(***************************判断纠偏从轴1是否超限********************************)	
AxisRecDevPos_H:=arrAxisPar[SlaveNo1].arrTargetPoint[0]-AxisPos_H;//轴纠偏上限
AxisRecDevPos_L:=arrAxisPar[SlaveNo1].arrTargetPoint[0]-AxisPos_L;//轴纠偏下限
AxisRecDevActPos1:=REAL_TO_LREAL(arrAxisCtrl[SlaveNo1].Status.fActPos);
IF AxisRecDevActPos1 > AxisRecDevPos_H OR AxisRecDevActPos1 < AxisRecDevPos_L THEN
	PosOverLimit1:=TRUE;//纠偏超限
ELSE
	PosOverLimit1:=FALSE;
END_IF
(***************************判断纠偏从轴2是否超限********************************)	
AxisRecDevPos_H:=arrAxisPar[SlaveNo2].arrTargetPoint[0]-AxisPos_H;//轴纠偏上限
AxisRecDevPos_L:=arrAxisPar[SlaveNo2].arrTargetPoint[0]-AxisPos_L;//轴纠偏下限
AxisRecDevActPos2:=REAL_TO_LREAL(arrAxisCtrl[SlaveNo2].Status.fActPos);
IF AxisRecDevActPos2 > AxisRecDevPos_H OR AxisRecDevActPos2 < AxisRecDevPos_L THEN
	PosOverLimit1:=TRUE;//纠偏超限
ELSE
	PosOverLimit1:=FALSE;
END_IF

IF Enable THEN
	CASE Step0 OF
		0://判断凸轮是否耦合
			IF NOT TON2.Q THEN
				TON2.IN:=TRUE;
				IF arrAxisCtrl[SlaveNo1].Status.Coupled AND arrAxisCtrl[SlaveNo2].Status.Coupled  THEN
					TON2.IN:=FALSE;
					Step0:=10;					
				END_IF
			ELSE
					TON2.IN:=FALSE;
					Error[0]:=TRUE;//纠偏凸轮耦合失败
					Step0:=9999;	//报警	
			END_IF
		10://判断主轴是是否启动，没启动则启动主轴
				IF arrAxisCtrl[MasterNo].Status.fActVelo>0 THEN
					Step0:=20;
				ELSE
					arrAxisCtrl[MasterNo].Cmd.bEnable:=TRUE;
					IF arrAxisCtrl[MasterNo].Status.Enabled THEN
						arrAxisPar[MasterNo].fVelocity_of_Velo:=MasterValue;//主轴速度
						arrAxisCtrl[MasterNo].Cmd.bMoveVelo:=TRUE;//主轴匀速启动							
					END_IF
				END_IF
		20://从轴纠偏速度计算
				TON1.IN:=TRUE;		
				IF RecDevPV > RecDevSensors_H AND TON1.Q THEN //纠偏传感器的当前值 大于 纠偏上限 
					IF NOT PosOverLimit1 AND NOT  PosOverLimit2 AND  arrAxisCtrl[SlaveNo1].Io.biNegLimit  AND  arrAxisCtrl[SlaveNo2].Io.biNegLimit  THEN//判断纠偏是否超限
						MC_RecDevvelocity_M:=(RecDevPV-RecDevSensors_H)*RecDevSpeedCoe;
						IF NOT CWW THEN
							MC_RecDevvelocity:=ScaleTrans(EN:=TRUE , Scalln:=MC_RecDevvelocity_M , X0:=0 , Y0:=0 , X1:=400 , Y1:=10 , Sclofs:=0 );//ScaleTrans的作用是将X0至X1范围之间的输入值，转换为Y0至Y1范围之间的输出值
						ELSE
							MC_RecDevvelocity:=-ScaleTrans(EN:=TRUE , Scalln:=MC_RecDevvelocity_M , X0:=0 , Y0:=0 , X1:=400 , Y1:=10 , Sclofs:=0 );
						END_IF
					ELSE
						Error[1]:=TRUE;//纠偏负限位报警
						MC_RecDevvelocity:=0;
					END_IF
				ELSIF RecDevPV < RecDevSensors_L AND TON1.Q  THEN//纠偏传感器的当前值 小于 纠偏下限
					IF NOT PosOverLimit1 AND NOT PosOverLimit2 AND  arrAxisCtrl[SlaveNo1].Io.biPosLimit AND  arrAxisCtrl[SlaveNo2].Io.biPosLimit  THEN
						MC_RecDevvelocity_M:=(RecDevSensors_L-RecDevPV)*RecDevSpeedCoe;//判断纠偏是否超限
						IF NOT CWW THEN
							MC_RecDevvelocity:=-ScaleTrans(EN:=TRUE , Scalln:=MC_RecDevvelocity_M , X0:=0 , Y0:=0 , X1:=400 , Y1:=10 , Sclofs:=0 );
						ELSE
							MC_RecDevvelocity:=ScaleTrans(EN:=TRUE , Scalln:=MC_RecDevvelocity_M , X0:=0 , Y0:=0 , X1:=400 , Y1:=10 , Sclofs:=0 );
						END_IF	
					ELSE
						Error[2]:=TRUE;//纠偏正限位报警
						MC_RecDevvelocity:=0;
					END_IF	
				ELSE
					MC_RecDevvelocity:=0;		
				END_IF					
	END_CASE
ELSE
		MC_RecDevvelocity:=0;//从轴的纠偏速度
		Step0:=0;
		TON1.IN:=FALSE;
		TON2.IN:=FALSE;
		IF RestHMI THEN
			Error[0]:=FALSE;//纠偏凸轮耦合失败
			Error[1]:=FALSE;//纠偏负限位报警
			Error[2]:=FALSE;//纠偏正限位报警
		END_IF
END_IF	
//纠偏齿轮耦合
IF MasterValue<>0 THEN
	GearInMultiMaster.GearRatio1:=MC_RecDevvelocity/MasterValue;
ELSE
	GearInMultiMaster.GearRatio1:=0;
END_IF
//多主轴耦合，不管主轴的停止还是运行中，都可以耦合从轴
GearInMultiMaster(
	Master1:=arrAxis[MasterNo] , 
	Master2:=arrAxis[SlaveNo1] , 
	Master3:=arrAxis[SlaveNo1] , 
	Master4:=arrAxis[SlaveNo1] , 
	Slave:=arrAxis[SlaveNo1]  , 
	Enable:=Enable , 
	GearRatio1:= , 
	GearRatio2:=0 , 
	GearRatio3:=0 , 
	GearRatio4:=0 , 
	Acceleration:= , 
	Deceleration:= , 
	Jerk:= , 
	BufferMode:= , 
	Options:= , 
	InGear=> , 
	Busy=> , 
	Active=> , 
	CommandAborted=> , 
	Error=> , 
	ErrorID=> );
//多主轴耦合，不管主轴的停止还是运行中，都可以耦合从轴
GearInMultiMaster1(
	Master1:=arrAxis[SlaveNo1] , 
	Master2:=arrAxis[SlaveNo2] , 
	Master3:=arrAxis[SlaveNo2] , 
	Master4:=arrAxis[SlaveNo2] , 
	Slave:=arrAxis[SlaveNo2]  , 
	Enable:=Enable , 
	GearRatio1:=1 , 
	GearRatio2:=0 , 
	GearRatio3:=0 , 
	GearRatio4:=0 , 
	Acceleration:= , 
	Deceleration:= , 
	Jerk:= , 
	BufferMode:= , 
	Options:= , 
	InGear=> , 
	Busy=> , 
	Active=> , 
	CommandAborted=> , 
	Error=> , 
	ErrorID=> );	
//纠偏从轴1解耦
SlaveCamOut(
	Slave:=arrAxis[SlaveNo1] , 
	Execute:=sF_TRIG.Q OR sR_TRIG.Q , 
	Options:= , 
	Done=> , 
	Busy=> , 
	Error=> , 
	ErrorID=> );
	//纠偏从轴2解耦
SlaveCamOut2(
	Slave:=arrAxis[SlaveNo2] , 
	Execute:=sF_TRIG.Q OR sR_TRIG.Q , 
	Options:= , 
	Done=> , 
	Busy=> , 
	Error=> , 
	ErrorID=> );
//从轴1停止
Slave_Stop(
	Axis:=arrAxis[SlaveNo1] , 
	Execute:=sF_TRIG.Q   , 
	Deceleration:= , 
	Jerk:= , 
	Options:= , 
	Done=> , 
	Busy=> , 
	Active=> , 
	CommandAborted=> , 
	Error=> , 
	ErrorID=> );
//从轴2停止
Slave_Stop2(
	Axis:=arrAxis[SlaveNo2] , 
	Execute:=sF_TRIG.Q   , 
	Deceleration:= , 
	Jerk:= , 
	Options:= , 
	Done=> , 
	Busy=> , 
	Active=> , 
	CommandAborted=> , 
	Error=> , 
	ErrorID=> );

END_FUNCTION_BLOCK

// ---- P2POUs/BasicFunction/01_IO/ScaleTrans.TcPOU
FUNCTION ScaleTrans : REAL
VAR_INPUT
	EN:BOOL;//启动条件
	Scalln:REAL;//输入值
	X0:REAL;//输入范围下限值
	Y0:REAL;//输出范围下限值
	X1:REAL;//输入范围上限值
	Y1:REAL;//输出范围上限值
	Sclofs:REAL;//偏置值
END_VAR
VAR
END_VAR

IF EN THEN
	IF (X1-X0)<> 0 THEN
		ScaleTrans:=(Y1-Y0)/(X1-X0)*(Scalln-X0)+Y0+Sclofs;
	END_IF
END_IF

END_FUNCTION

// ---- P2POUs/BasicFunction/12_User2/FB_BlueGlue.TcPOU
FUNCTION_BLOCK FB_BlueGlue//蓝胶检测自动
VAR_INPUT
	Enable:BOOL;//启动条件
	BlueSenser:BOOL;//蓝胶检测信号
	An_Quantited:UINT;//正极已叠片极片数
	An_QuantitSet:UINT;//正极设定叠片片
	Ca_Quantited:UINT;//负极已叠片极片数
	Ca_QuantitSet:UINT;//负极设定叠片片
	Distance:REAL;//蓝胶检测Semer到压刀的距离
	BluWidth:REAL;//蓝胶宽度
	Width:REAL;//压刀外边距宽度	 
END_VAR
VAR_OUTPUT
END_VAR
VAR_IN_OUT
		BluGlueNG:ARRAY[0..1] OF BOOL;
END_VAR
VAR
	// 正、负极已叠极片总数
	Quantited: UINT;
	// 正、负极设定极片总数
	QuantitSet: UINT;
	// 正、负极未叠片数
	Quantit: UINT;
	// 未叠极片所需隔膜长度
	Distance_DT: REAL;
	// 蓝胶到压刀距离上限
	Distance_H: REAL;
	// 蓝胶到压针距离下限
	Distance_L: REAL;
	Step0: INT;

	blue_R_TRIG: R_TRIG;
	blue_F_TRIG: F_TRIG;
END_VAR

//计算已叠极片总数
Quantited:=An_Quantited+Ca_Quantited;
//计算正、负极片设定总数
QuantitSet:=An_QuantitSet+Ca_QuantitSet;
//计算未叠片数
Quantit:=QuantitSet-Quantited;
//未叠正、负极片所需隔膜总长度
Distance_DT:=Width*Quantit;
//蓝胶到压针距离上限
Distance_H:=Distance+BluWidth+10;
//蓝胶到压针距离下降
Distance_L:=Distance+BluWidth-10;
//蓝胶检测信号上升沿
blue_R_TRIG(CLK:=BlueSenser, Q=> );
//蓝胶要信号下降沿
blue_F_TRIG(CLK:=BlueSenser , Q=> );
IF Enable THEN
	CASE Step0 OF
			0://判断是否检测到蓝胶信号
				IF blue_R_TRIG.Q THEN
					Step0:=10;
				END_IF
			10://根据未叠片隔膜长度与蓝胶到压刀的距离判断是当前电芯NG、下一个电芯NG、当前以及下一个电芯都NG
				IF  Distance_DT<Distance_L THEN //未叠片隔膜长度小于蓝胶所需隔膜长度下限，下一个电芯NG
					BluGlueNG[1]:=TRUE;
					Step0:=20;
				ELSIF Distance_DT>Distance_L AND Distance_DT< Distance_H  THEN//未叠片隔膜长度在蓝胶上、下限之间，则当前电芯、下个电芯都NG
					BluGlueNG[0]:=TRUE;
					BluGlueNG[1]:=TRUE;
					Step0:=20;
				ELSIF Distance_DT> Distance_H THEN//未叠片隔膜长度大于蓝胶所需隔膜长度上限，当前电芯NG
					BluGlueNG[0]:=TRUE;
					Step0:=20;
				END_IF
			20://判断检测是否结束
				IF blue_F_TRIG.Q THEN
					Step0:=0;
				END_IF
	END_CASE
END_IF

END_FUNCTION_BLOCK

// ---- P2POUs/BasicFunction/12_User2/FB_Demarcate.TcPOU
FUNCTION_BLOCK FB_Demarcate//CCD标定自动程序
VAR_INPUT
	AxisX1_NO : INT; //X1轴号
	AxisX2_NO : INT;//X2轴号
	AxisY_NO  : INT;//Y轴号	
END_VAR
VAR_OUTPUT
	
END_VAR
VAR
	
	i: INT;
	// 拍照延时复位
	TON1: TON;
	TON2: TON;
	// CCD标定上升沿
	rCCD_Demarcate: R_TRIG;
	singeMode: BOOL;
	singeStep0: BOOL;
	fCCD_Demarcate: F_TRIG;
	bTest1: BOOL;
	iTest: INT;
END_VAR

VAR_IN_OUT
	Step0: INT;//程序步
	DemarcateStart:BOOL;//CCD标定启动	
	CCDStart: BOOL;// CCD拍照启动
	CCDNo:INT;//ccd拍照次数记数
	DemarcateResult:INT;//标定结果
	DemarcateDone: BOOL;	// CCD标定完成
	Demarcateing: BOOL;	// CCD标定中
	// CCD标定NG报警
	Error: BOOL;
END_VAR

TON1(IN:= , PT:=T#2S , Q=> , ET=> );//拍照延时复位
TON2(IN:= , PT:=T#0.2S , Q=> , ET=> );//拍照延时
rCCD_Demarcate(CLK:=DemarcateStart , Q=> );//CCD标定启动上升沿
fCCD_Demarcate(CLK:=DemarcateStart , Q=> );//CCD标定启动上升沿
IF rCCD_Demarcate.Q THEN
	Error:=FALSE;//CCD标定NG报警
	TON1.IN:=FALSE;
	Step0:=0;
END_IF



CASE Step0 OF
		0://等待CCD标定启动信号
			IF fCCD_Demarcate.Q THEN
						i:=0;//标定点位记数
						TON1.IN:=FALSE;
						DemarcateStart:=FALSE;//复位标定启动
						DemarcateDone:=FALSE;//CCD标定完成
						Demarcateing:=TRUE;//CCD标定中
						IF singeMode THEN
							singeStep0:=TRUE;
						ELSE
							singeStep0:=FALSE;
						END_IF
						Step0:=10;
			END_IF
	10://X1、X2先回初始位
				IF  NOT singeStep0 THEN
							TON1.IN:=FALSE;
							IF arrAxisCtrl[AxisX1_NO].Status.Homed AND arrAxisCtrl[AxisX1_NO].Status.NoMoving THEN
										IF arrAxisCtrl[AxisX1_NO].Cmd.arrbRealPoint[1] THEN
											arrAxisCtrl[AxisX1_NO].Cmd.iGoSetPos:=0;
										ELSE
											arrAxisCtrl[AxisX1_NO].Cmd.iGoSetPos:=1;
										END_IF
							END_IF
							IF arrAxisCtrl[AxisX2_NO].Status.Homed AND arrAxisCtrl[AxisX2_NO].Status.NoMoving  THEN
										IF arrAxisCtrl[AxisX2_NO].Cmd.arrbRealPoint[1] THEN
											arrAxisCtrl[AxisX2_NO].Cmd.iGoSetPos:=0;
										ELSE
											arrAxisCtrl[AxisX2_NO].Cmd.iGoSetPos:=1;
										END_IF
							END_IF	
							IF  arrAxisCtrl[AxisX1_NO].Cmd.arrbRealPoint[1]  AND 	arrAxisCtrl[AxisX2_NO].Cmd.arrbRealPoint[1]THEN
								IF singeMode THEN
									singeStep0:=TRUE;
								ELSE
									singeStep0:=FALSE;
								END_IF
								Step0:=11;
							END_IF	
				END_IF		
	11://Y回初始位
				IF NOT singeStep0 THEN
									IF arrAxisCtrl[AxisY_NO].Status.Homed AND arrAxisCtrl[AxisY_NO].Status.NoMoving  THEN
											IF arrAxisCtrl[AxisY_NO].Cmd.arrbRealPoint[1] THEN
												arrAxisCtrl[AxisY_NO].Cmd.iGoSetPos:=0;
													IF singeMode THEN
														singeStep0:=TRUE;
													ELSE
														singeStep0:=FALSE;
													END_IF
													Step0:=12;									
											ELSE
												arrAxisCtrl[AxisY_NO].Cmd.iGoSetPos:=1;
											END_IF
								END_IF
				END_IF			
		12://判断CCD标定走到第几个点位
						IF NOT  singeStep0 THEN
											DemarcateResult:=0;
											IF  i=0    THEN//(-4,-4)
															arrAxisPar[AxisX1_NO].arrTargetPoint[3]:=arrAxisPar[AxisX1_NO].arrTargetPoint[1]-4;//+(103.94*COS(DEG_TO_RAD(CCD_W+225))-103.94*COS(DEG_TO_RAD(225))); 
															arrAxisPar[AxisX2_NO].arrTargetPoint[3]:=arrAxisPar[AxisX2_NO].arrTargetPoint[1]-4;//+(103.94*SIN(DEG_TO_RAD(CCD_W+315))-103.94*COS(DEG_TO_RAD(315)));
															arrAxisPar[AxisY_NO].arrTargetPoint[3]:=arrAxisPar[AxisY_NO].arrTargetPoint[1]-4;//+(103.94*COS(DEG_TO_RAD(CCD_W+135))-103.94*COS(DEG_TO_RAD(135)));	
															i:=i+1;
															IF singeMode THEN
																singeStep0:=TRUE;
															ELSE
																singeStep0:=FALSE;
															END_IF
															Step0:=20;
											ELSIF i=1 THEN//(0,-4)
															arrAxisPar[AxisX1_NO].arrTargetPoint[3]:=arrAxisPar[AxisX1_NO].arrTargetPoint[1];//+(103.94*COS(DEG_TO_RAD(CCD_W+225))-103.94*COS(DEG_TO_RAD(225))); 
															arrAxisPar[AxisX2_NO].arrTargetPoint[3]:=arrAxisPar[AxisX2_NO].arrTargetPoint[1];//+(103.94*SIN(DEG_TO_RAD(CCD_W+315))-103.94*COS(DEG_TO_RAD(315)));
															arrAxisPar[AxisY_NO].arrTargetPoint[3]:=arrAxisPar[AxisY_NO].arrTargetPoint[1]-4;//+(103.94*COS(DEG_TO_RAD(CCD_W+135))-103.94*COS(DEG_TO_RAD(135)));
															i:=i+1;
															IF singeMode THEN
																singeStep0:=TRUE;
															ELSE
																singeStep0:=FALSE;
															END_IF
															Step0:=20;
											ELSIF i=2 THEN//(4,-4)
															arrAxisPar[AxisX1_NO].arrTargetPoint[3]:=arrAxisPar[AxisX1_NO].arrTargetPoint[1]+4;//+(103.94*COS(DEG_TO_RAD(CCD_W+225))-103.94*COS(DEG_TO_RAD(225))); 
															arrAxisPar[AxisX2_NO].arrTargetPoint[3]:=arrAxisPar[AxisX2_NO].arrTargetPoint[1]+4;//+(103.94*SIN(DEG_TO_RAD(CCD_W+315))-103.94*COS(DEG_TO_RAD(315)));
															arrAxisPar[AxisY_NO].arrTargetPoint[3]:=arrAxisPar[AxisY_NO].arrTargetPoint[1]-4;//+(103.94*COS(DEG_TO_RAD(CCD_W+135))-103.94*COS(DEG_TO_RAD(135)));	
															i:=i+1;
															IF singeMode THEN
																singeStep0:=TRUE;
															ELSE
																singeStep0:=FALSE;
															END_IF
															Step0:=20;									
											ELSIF i=3 THEN//(4,0)
														arrAxisPar[AxisX1_NO].arrTargetPoint[3]:=arrAxisPar[AxisX1_NO].arrTargetPoint[1]+4;//+(103.94*COS(DEG_TO_RAD(CCD_W+225))-103.94*COS(DEG_TO_RAD(225))); 
														arrAxisPar[AxisX2_NO].arrTargetPoint[3]:=arrAxisPar[AxisX2_NO].arrTargetPoint[1]+4;//+(103.94*SIN(DEG_TO_RAD(CCD_W+315))-103.94*COS(DEG_TO_RAD(315)));
														arrAxisPar[AxisY_NO].arrTargetPoint[3]:=arrAxisPar[AxisY_NO].arrTargetPoint[1];//+(103.94*COS(DEG_TO_RAD(CCD_W+135))-103.94*COS(DEG_TO_RAD(135)));	
														i:=i+1;
														IF singeMode THEN
																singeStep0:=TRUE;
															ELSE
																singeStep0:=FALSE;
															END_IF
														Step0:=20;		
											ELSIF i=4 THEN//(0,0)
														arrAxisPar[AxisX1_NO].arrTargetPoint[3]:=arrAxisPar[AxisX1_NO].arrTargetPoint[1];//+(103.94*COS(DEG_TO_RAD(CCD_W+225))-103.94*COS(DEG_TO_RAD(225))); 
														arrAxisPar[AxisX2_NO].arrTargetPoint[3]:=arrAxisPar[AxisX2_NO].arrTargetPoint[1];//+(103.94*SIN(DEG_TO_RAD(CCD_W+315))-103.94*COS(DEG_TO_RAD(315)));
														arrAxisPar[AxisY_NO].arrTargetPoint[3]:=arrAxisPar[AxisY_NO].arrTargetPoint[1];//+(103.94*COS(DEG_TO_RAD(CCD_W+135))-103.94*COS(DEG_TO_RAD(135)));	
														i:=i+1;
														Step0:=20;		
											ELSIF i=5 THEN//(-4,0)
														arrAxisPar[AxisX1_NO].arrTargetPoint[3]:=arrAxisPar[AxisX1_NO].arrTargetPoint[1]-4;//+(103.94*COS(DEG_TO_RAD(CCD_W+225))-103.94*COS(DEG_TO_RAD(225))); 
														arrAxisPar[AxisX2_NO].arrTargetPoint[3]:=arrAxisPar[AxisX2_NO].arrTargetPoint[1]-4;//+(103.94*SIN(DEG_TO_RAD(CCD_W+315))-103.94*COS(DEG_TO_RAD(315)));
														arrAxisPar[AxisY_NO].arrTargetPoint[3]:=arrAxisPar[AxisY_NO].arrTargetPoint[1];//+(103.94*COS(DEG_TO_RAD(CCD_W+135))-103.94*COS(DEG_TO_RAD(135)));	
														i:=i+1;
														IF singeMode THEN
																singeStep0:=TRUE;
															ELSE
																singeStep0:=FALSE;
															END_IF
														Step0:=20;		
											ELSIF i=6 THEN//(-4,4)
															arrAxisPar[AxisX1_NO].arrTargetPoint[3]:=arrAxisPar[AxisX1_NO].arrTargetPoint[1]-4;//+(103.94*COS(DEG_TO_RAD(CCD_W+225))-103.94*COS(DEG_TO_RAD(225))); 
															arrAxisPar[AxisX2_NO].arrTargetPoint[3]:=arrAxisPar[AxisX2_NO].arrTargetPoint[1]-4;//+(103.94*SIN(DEG_TO_RAD(CCD_W+315))-103.94*COS(DEG_TO_RAD(315)));
															arrAxisPar[AxisY_NO].arrTargetPoint[3]:=arrAxisPar[AxisY_NO].arrTargetPoint[1]+4;//+(103.94*COS(DEG_TO_RAD(CCD_W+135))-103.94*COS(DEG_TO_RAD(135)));
															i:=i+1;
															IF singeMode THEN
																singeStep0:=TRUE;
															ELSE
																singeStep0:=FALSE;
															END_IF
															Step0:=20;		
											ELSIF i=7 THEN//(0,4)
															arrAxisPar[AxisX1_NO].arrTargetPoint[3]:=arrAxisPar[AxisX1_NO].arrTargetPoint[1];//+(103.94*COS(DEG_TO_RAD(CCD_W+225))-103.94*COS(DEG_TO_RAD(225))); 
															arrAxisPar[AxisX2_NO].arrTargetPoint[3]:=arrAxisPar[AxisX2_NO].arrTargetPoint[1];//+(103.94*SIN(DEG_TO_RAD(CCD_W+315))-103.94*COS(DEG_TO_RAD(315)));
															arrAxisPar[AxisY_NO].arrTargetPoint[3]:=arrAxisPar[AxisY_NO].arrTargetPoint[1]+4;//+(103.94*COS(DEG_TO_RAD(CCD_W+135))-103.94*COS(DEG_TO_RAD(135)));	
															i:=i+1;
															IF singeMode THEN
																singeStep0:=TRUE;
															ELSE
																singeStep0:=FALSE;
															END_IF
															Step0:=20;		
											ELSIF i=8 THEN//(4,4)
														arrAxisPar[AxisX1_NO].arrTargetPoint[3]:=arrAxisPar[AxisX1_NO].arrTargetPoint[1]+4;//+(103.94*COS(DEG_TO_RAD(CCD_W+225))-103.94*COS(DEG_TO_RAD(225))); 
														arrAxisPar[AxisX2_NO].arrTargetPoint[3]:=arrAxisPar[AxisX2_NO].arrTargetPoint[1]+4;//+(103.94*SIN(DEG_TO_RAD(CCD_W+315))-103.94*COS(DEG_TO_RAD(315)));
														arrAxisPar[AxisY_NO].arrTargetPoint[3]:=arrAxisPar[AxisY_NO].arrTargetPoint[1]+4;//+(103.94*COS(DEG_TO_RAD(CCD_W+135))-103.94*COS(DEG_TO_RAD(135)));	
														i:=i+1;
														IF singeMode THEN
																singeStep0:=TRUE;
															ELSE
																singeStep0:=FALSE;
															END_IF
														Step0:=20;		
											ELSIF i=9 THEN//(0,0,-2)
														arrAxisPar[AxisX1_NO].arrTargetPoint[3]:=arrAxisPar[AxisX1_NO].arrTargetPoint[1]+(103.94*COS(DEG_TO_RAD(-2+225))-103.94*COS(DEG_TO_RAD(225))); 
														arrAxisPar[AxisX2_NO].arrTargetPoint[3]:=arrAxisPar[AxisX2_NO].arrTargetPoint[1]+(103.94*COS(DEG_TO_RAD(-2+135))-103.94*COS(DEG_TO_RAD(135)));
														arrAxisPar[AxisY_NO].arrTargetPoint[3]:=arrAxisPar[AxisY_NO].arrTargetPoint[1]+(103.94*SIN(DEG_TO_RAD(-2+315))-103.94*SIN(DEG_TO_RAD(315)));	
														i:=i+1;
														IF singeMode THEN
																singeStep0:=TRUE;
															ELSE
																singeStep0:=FALSE;
															END_IF
														Step0:=20;		
											ELSIF i=10 THEN//(0,0)
														arrAxisPar[AxisX1_NO].arrTargetPoint[3]:=arrAxisPar[AxisX1_NO].arrTargetPoint[1];//+(103.94*COS(DEG_TO_RAD(2+225))-103.94*COS(DEG_TO_RAD(225))); 
														arrAxisPar[AxisX2_NO].arrTargetPoint[3]:=arrAxisPar[AxisX2_NO].arrTargetPoint[1];//+(103.94*SIN(DEG_TO_RAD(2+315))-103.94*COS(DEG_TO_RAD(315)));
														arrAxisPar[AxisY_NO].arrTargetPoint[3]:=arrAxisPar[AxisY_NO].arrTargetPoint[1];//+(103.94*COS(DEG_TO_RAD(2+135))-103.94*COS(DEG_TO_RAD(135)));	
														i:=i+1;
														IF singeMode THEN
																singeStep0:=TRUE;
															ELSE
																singeStep0:=FALSE;
															END_IF
														Step0:=20;		
											ELSIF i=11  THEN//(0,0,2)
															arrAxisPar[AxisX1_NO].arrTargetPoint[3]:=arrAxisPar[AxisX1_NO].arrTargetPoint[1]+(103.94*COS(DEG_TO_RAD(2+225))-103.94*COS(DEG_TO_RAD(225))); 
															arrAxisPar[AxisX2_NO].arrTargetPoint[3]:=arrAxisPar[AxisX2_NO].arrTargetPoint[1]+(103.94*COS(DEG_TO_RAD(2+135))-103.94*COS(DEG_TO_RAD(135)));
															arrAxisPar[AxisY_NO].arrTargetPoint[3]:=arrAxisPar[AxisY_NO].arrTargetPoint[1]+(103.94*SIN(DEG_TO_RAD(2+315))-103.94*SIN(DEG_TO_RAD(315)));
															i:=i+1;
															IF singeMode THEN
																singeStep0:=TRUE;
															ELSE
																singeStep0:=FALSE;
															END_IF
															Step0:=20;		
											ELSIF i=130 THEN
															arrAxisPar[AxisX1_NO].arrTargetPoint[3]:=arrAxisPar[AxisX1_NO].arrTargetPoint[1];//+(103.94*COS(DEG_TO_RAD(CCD_W+225))-103.94*COS(DEG_TO_RAD(225))); 
															arrAxisPar[AxisX2_NO].arrTargetPoint[3]:=arrAxisPar[AxisX2_NO].arrTargetPoint[1];//+(103.94*SIN(DEG_TO_RAD(CCD_W+315))-103.94*COS(DEG_TO_RAD(315)));
															arrAxisPar[AxisY_NO].arrTargetPoint[3]:=arrAxisPar[AxisY_NO].arrTargetPoint[1];//+(103.94*COS(DEG_TO_RAD(CCD_W+135))-103.94*COS(DEG_TO_RAD(135)));	
															i:=i+1;
															IF singeMode THEN
																singeStep0:=TRUE;
															ELSE
																singeStep0:=FALSE;
															END_IF
															Step0:=20;		
											ELSIF i=140 THEN
														arrAxisPar[AxisX1_NO].arrTargetPoint[3]:=arrAxisPar[AxisX1_NO].arrTargetPoint[1]+(103.94*COS(DEG_TO_RAD(-1+225))-103.94*COS(DEG_TO_RAD(225))); 
														arrAxisPar[AxisX2_NO].arrTargetPoint[3]:=arrAxisPar[AxisX2_NO].arrTargetPoint[1]+(103.94*SIN(DEG_TO_RAD(-1+315))-103.94*COS(DEG_TO_RAD(315)));
														arrAxisPar[AxisY_NO].arrTargetPoint[3]:=arrAxisPar[AxisY_NO].arrTargetPoint[1]+(103.94*COS(DEG_TO_RAD(-1+135))-103.94*COS(DEG_TO_RAD(135)));	
														i:=i+1;
														IF singeMode THEN
																singeStep0:=TRUE;
															ELSE
																singeStep0:=FALSE;
															END_IF
														Step0:=20;		
											ELSIF i=150 THEN
														arrAxisPar[AxisX1_NO].arrTargetPoint[3]:=arrAxisPar[AxisX1_NO].arrTargetPoint[1]+(103.94*COS(DEG_TO_RAD(-2+225))-103.94*COS(DEG_TO_RAD(225))); 
														arrAxisPar[AxisX2_NO].arrTargetPoint[3]:=arrAxisPar[AxisX2_NO].arrTargetPoint[1]+(103.94*SIN(DEG_TO_RAD(-2+315))-103.94*COS(DEG_TO_RAD(315)));
														arrAxisPar[AxisY_NO].arrTargetPoint[3]:=arrAxisPar[AxisY_NO].arrTargetPoint[1]+(103.94*COS(DEG_TO_RAD(-2+135))-103.94*COS(DEG_TO_RAD(135)));	
														i:=i+1;
														IF singeMode THEN
																singeStep0:=TRUE;
															ELSE
																singeStep0:=FALSE;
															END_IF
														Step0:=20;		
											ELSIF i=160 THEN
														arrAxisPar[AxisX1_NO].arrTargetPoint[3]:=arrAxisPar[AxisX1_NO].arrTargetPoint[1];//+(103.94*COS(DEG_TO_RAD(CCD_W+225))-103.94*COS(DEG_TO_RAD(225))); 
														arrAxisPar[AxisX2_NO].arrTargetPoint[3]:=arrAxisPar[AxisX2_NO].arrTargetPoint[1];//+(103.94*SIN(DEG_TO_RAD(CCD_W+315))-103.94*COS(DEG_TO_RAD(315)));
														arrAxisPar[AxisY_NO].arrTargetPoint[3]:=arrAxisPar[AxisY_NO].arrTargetPoint[1];//+(103.94*COS(DEG_TO_RAD(CCD_W+135))-103.94*COS(DEG_TO_RAD(135)));		
														i:=i+1;
														Step0:=20;													
											END_IF
						END_IF	
	20://先移动X1,X2
				IF  NOT singeStep0 THEN
					IF NOT TON1.Q THEN
										TON1.IN:=TRUE;
					ELSE
										IF arrAxisCtrl[AxisX1_NO].Status.Homed AND arrAxisCtrl[AxisX1_NO].Status.NoMoving THEN
													IF arrAxisCtrl[AxisX1_NO].Cmd.arrbRealPoint[3] THEN
														arrAxisCtrl[AxisX1_NO].Cmd.iGoSetPos:=0;
													ELSE
														arrAxisCtrl[AxisX1_NO].Cmd.iGoSetPos:=3;
													END_IF
										END_IF
										IF arrAxisCtrl[AxisX2_NO].Status.Homed AND arrAxisCtrl[AxisX2_NO].Status.NoMoving  THEN
													IF arrAxisCtrl[AxisX2_NO].Cmd.arrbRealPoint[3] THEN
														arrAxisCtrl[AxisX2_NO].Cmd.iGoSetPos:=0;
													ELSE
														arrAxisCtrl[AxisX2_NO].Cmd.iGoSetPos:=3;
													END_IF
										END_IF	
										IF  arrAxisCtrl[AxisX1_NO].Cmd.arrbRealPoint[3]  AND arrAxisCtrl[AxisX1_NO].Status.NoMoving AND 
							 				arrAxisCtrl[AxisX2_NO].Cmd.arrbRealPoint[3] AND arrAxisCtrl[AxisX2_NO].Status.NoMoving THEN
													IF singeMode THEN
														singeStep0:=TRUE;
													ELSE
														singeStep0:=FALSE;
													END_IF
													TON1.IN:=FALSE;
													Step0:=30;
										ELSIF arrAxisCtrl[AxisX1_NO].Status.Error OR arrAxisCtrl[AxisX2_NO].Status.Error THEN
													TON1.IN:=FALSE;
													Step0:=0;											
										END_IF	
						END_IF
				END_IF	
	30://再移动Y
				IF NOT singeStep0 THEN
							IF NOT TON1.Q THEN
										TON1.IN:=TRUE;
							ELSE
									IF arrAxisCtrl[AxisY_NO].Status.Homed AND arrAxisCtrl[AxisY_NO].Status.NoMoving  THEN
												IF arrAxisCtrl[AxisY_NO].Cmd.arrbRealPoint[3] THEN
													arrAxisCtrl[AxisY_NO].Cmd.iGoSetPos:=0;
														IF singeMode THEN
															singeStep0:=TRUE;
														ELSE
															singeStep0:=FALSE;
														END_IF
														TON1.IN:=FALSE;
														 TON2.IN:=FALSE;
														Step0:=31;									
												ELSE
													arrAxisCtrl[AxisY_NO].Cmd.iGoSetPos:=3;
												END_IF
								ELSIF   arrAxisCtrl[AxisY_NO].Status.Error THEN
														TON1.IN:=FALSE;
														Step0:=0;										
								END_IF
							END_IF
				END_IF
				
	31:
	    TON2.IN:=TRUE;
		IF TON2.Q THEN
				CCDNo:=i;
				CCDStart:=TRUE;
				DemarcateResult:=0;	
				Step0:=40;	
				 TON2.IN:=FALSE;
		END_IF		 
	40://启动拍照
			IF NOT TON1.Q THEN
				TON1.IN:=TRUE;
			ELSE
				TON1.IN:=FALSE;	
				CCDStart:=FALSE;
				Step0:=50;
			END_IF
	50://等待标定结果
			IF DemarcateResult=1 THEN
				DemarcateResult:=0; 
				 Step0:=60;
			ELSE
				Error:=TRUE;//CCD标定NG报警
				Step0:=9999;
			END_IF
	60://判断标定次数
			IF i>=12 THEN
				Step0:=0;
				Demarcateing:=FALSE;
			ELSE
				Step0:=10;
			END_IF				
END_CASE







IF bTest1 THEN
	
   CASE iTest OF
	 0://(-4,-4)
				arrAxisPar[AxisX1_NO].arrTargetPoint[3]:=arrAxisPar[AxisX1_NO].arrTargetPoint[1]-4;//+(103.94*COS(DEG_TO_RAD(CCD_W+225))-103.94*COS(DEG_TO_RAD(225))); 
				arrAxisPar[AxisX2_NO].arrTargetPoint[3]:=arrAxisPar[AxisX2_NO].arrTargetPoint[1]-4;//+(103.94*SIN(DEG_TO_RAD(CCD_W+315))-103.94*COS(DEG_TO_RAD(315)));
				arrAxisPar[AxisY_NO].arrTargetPoint[3]:=arrAxisPar[AxisY_NO].arrTargetPoint[1]-4;//+(103.94*COS(DEG_TO_RAD(CCD_W+135))-103.94*COS(DEG_TO_RAD(135)));	
				iTest:=50;
											
	 1://(0,-4)
			arrAxisPar[AxisX1_NO].arrTargetPoint[3]:=arrAxisPar[AxisX1_NO].arrTargetPoint[1];//+(103.94*COS(DEG_TO_RAD(CCD_W+225))-103.94*COS(DEG_TO_RAD(225))); 
		    arrAxisPar[AxisX2_NO].arrTargetPoint[3]:=arrAxisPar[AxisX2_NO].arrTargetPoint[1];//+(103.94*SIN(DEG_TO_RAD(CCD_W+315))-103.94*COS(DEG_TO_RAD(315)));
			arrAxisPar[AxisY_NO].arrTargetPoint[3]:=arrAxisPar[AxisY_NO].arrTargetPoint[1]-4;//+(103.94*COS(DEG_TO_RAD(CCD_W+135))-103.94*COS(DEG_TO_RAD(135)));
				iTest:=50;											
	2://(4,-4)
			arrAxisPar[AxisX1_NO].arrTargetPoint[3]:=arrAxisPar[AxisX1_NO].arrTargetPoint[1]+4;//+(103.94*COS(DEG_TO_RAD(CCD_W+225))-103.94*COS(DEG_TO_RAD(225))); 
			arrAxisPar[AxisX2_NO].arrTargetPoint[3]:=arrAxisPar[AxisX2_NO].arrTargetPoint[1]+4;//+(103.94*SIN(DEG_TO_RAD(CCD_W+315))-103.94*COS(DEG_TO_RAD(315)));
			arrAxisPar[AxisY_NO].arrTargetPoint[3]:=arrAxisPar[AxisY_NO].arrTargetPoint[1]-4;//+(103.94*COS(DEG_TO_RAD(CCD_W+135))-103.94*COS(DEG_TO_RAD(135)));	
				iTest:=50;															
	3://(4,0)
			arrAxisPar[AxisX1_NO].arrTargetPoint[3]:=arrAxisPar[AxisX1_NO].arrTargetPoint[1]+4;//+(103.94*COS(DEG_TO_RAD(CCD_W+225))-103.94*COS(DEG_TO_RAD(225))); 
			arrAxisPar[AxisX2_NO].arrTargetPoint[3]:=arrAxisPar[AxisX2_NO].arrTargetPoint[1]+4;//+(103.94*SIN(DEG_TO_RAD(CCD_W+315))-103.94*COS(DEG_TO_RAD(315)));
			arrAxisPar[AxisY_NO].arrTargetPoint[3]:=arrAxisPar[AxisY_NO].arrTargetPoint[1];//+(103.94*COS(DEG_TO_RAD(CCD_W+135))-103.94*COS(DEG_TO_RAD(135)));	
			iTest:=50;								
  4://(0,0)
		arrAxisPar[AxisX1_NO].arrTargetPoint[3]:=arrAxisPar[AxisX1_NO].arrTargetPoint[1];//+(103.94*COS(DEG_TO_RAD(CCD_W+225))-103.94*COS(DEG_TO_RAD(225))); 
		arrAxisPar[AxisX2_NO].arrTargetPoint[3]:=arrAxisPar[AxisX2_NO].arrTargetPoint[1];//+(103.94*SIN(DEG_TO_RAD(CCD_W+315))-103.94*COS(DEG_TO_RAD(315)));
			arrAxisPar[AxisY_NO].arrTargetPoint[3]:=arrAxisPar[AxisY_NO].arrTargetPoint[1];//+(103.94*COS(DEG_TO_RAD(CCD_W+135))-103.94*COS(DEG_TO_RAD(135)));	
			iTest:=50;
5://(-4,0)
			arrAxisPar[AxisX1_NO].arrTargetPoint[3]:=arrAxisPar[AxisX1_NO].arrTargetPoint[1]-4;//+(103.94*COS(DEG_TO_RAD(CCD_W+225))-103.94*COS(DEG_TO_RAD(225))); 
			arrAxisPar[AxisX2_NO].arrTargetPoint[3]:=arrAxisPar[AxisX2_NO].arrTargetPoint[1]-4;//+(103.94*SIN(DEG_TO_RAD(CCD_W+315))-103.94*COS(DEG_TO_RAD(315)));
		arrAxisPar[AxisY_NO].arrTargetPoint[3]:=arrAxisPar[AxisY_NO].arrTargetPoint[1];//+(103.94*COS(DEG_TO_RAD(CCD_W+135))-103.94*COS(DEG_TO_RAD(135)));	
		iTest:=50;
6://(-4,4)
			arrAxisPar[AxisX1_NO].arrTargetPoint[3]:=arrAxisPar[AxisX1_NO].arrTargetPoint[1]-4;//+(103.94*COS(DEG_TO_RAD(CCD_W+225))-103.94*COS(DEG_TO_RAD(225))); 
			arrAxisPar[AxisX2_NO].arrTargetPoint[3]:=arrAxisPar[AxisX2_NO].arrTargetPoint[1]-4;//+(103.94*SIN(DEG_TO_RAD(CCD_W+315))-103.94*COS(DEG_TO_RAD(315)));
			arrAxisPar[AxisY_NO].arrTargetPoint[3]:=arrAxisPar[AxisY_NO].arrTargetPoint[1]+4;//+(103.94*COS(DEG_TO_RAD(CCD_W+135))-103.94*COS(DEG_TO_RAD(135)));
			iTest:=50;										
7://(0,4)
		arrAxisPar[AxisX1_NO].arrTargetPoint[3]:=arrAxisPar[AxisX1_NO].arrTargetPoint[1];//+(103.94*COS(DEG_TO_RAD(CCD_W+225))-103.94*COS(DEG_TO_RAD(225))); 
		arrAxisPar[AxisX2_NO].arrTargetPoint[3]:=arrAxisPar[AxisX2_NO].arrTargetPoint[1];//+(103.94*SIN(DEG_TO_RAD(CCD_W+315))-103.94*COS(DEG_TO_RAD(315)));
		arrAxisPar[AxisY_NO].arrTargetPoint[3]:=arrAxisPar[AxisY_NO].arrTargetPoint[1]+4;//+(103.94*COS(DEG_TO_RAD(CCD_W+135))-103.94*COS(DEG_TO_RAD(135)));	
			iTest:=50;									
8://(4,4)
		arrAxisPar[AxisX1_NO].arrTargetPoint[3]:=arrAxisPar[AxisX1_NO].arrTargetPoint[1]+4;//+(103.94*COS(DEG_TO_RAD(CCD_W+225))-103.94*COS(DEG_TO_RAD(225))); 
			arrAxisPar[AxisX2_NO].arrTargetPoint[3]:=arrAxisPar[AxisX2_NO].arrTargetPoint[1]+4;//+(103.94*SIN(DEG_TO_RAD(CCD_W+315))-103.94*COS(DEG_TO_RAD(315)));
		arrAxisPar[AxisY_NO].arrTargetPoint[3]:=arrAxisPar[AxisY_NO].arrTargetPoint[1]+4;//+(103.94*COS(DEG_TO_RAD(CCD_W+135))-103.94*COS(DEG_TO_RAD(135)));	
		iTest:=50;
9://(0,0,-2)
			arrAxisPar[AxisX1_NO].arrTargetPoint[3]:=arrAxisPar[AxisX1_NO].arrTargetPoint[1]+(103.94*COS(DEG_TO_RAD(-2+225))-103.94*COS(DEG_TO_RAD(225))); 
				arrAxisPar[AxisX2_NO].arrTargetPoint[3]:=arrAxisPar[AxisX2_NO].arrTargetPoint[1]+(103.94*COS(DEG_TO_RAD(-2+135))-103.94*COS(DEG_TO_RAD(135)));
		arrAxisPar[AxisY_NO].arrTargetPoint[3]:=arrAxisPar[AxisY_NO].arrTargetPoint[1]+(103.94*SIN(DEG_TO_RAD(-2+315))-103.94*SIN(DEG_TO_RAD(315)));	
		iTest:=50;
11://(0,0,2)
				arrAxisPar[AxisX1_NO].arrTargetPoint[3]:=arrAxisPar[AxisX1_NO].arrTargetPoint[1]+(103.94*COS(DEG_TO_RAD(2+225))-103.94*COS(DEG_TO_RAD(225))); 
	arrAxisPar[AxisX2_NO].arrTargetPoint[3]:=arrAxisPar[AxisX2_NO].arrTargetPoint[1]+(103.94*COS(DEG_TO_RAD(2+135))-103.94*COS(DEG_TO_RAD(135)));
		arrAxisPar[AxisY_NO].arrTargetPoint[3]:=arrAxisPar[AxisY_NO].arrTargetPoint[1]+(103.94*SIN(DEG_TO_RAD(2+315))-103.94*SIN(DEG_TO_RAD(315)));
		iTest:=50;
12:
		arrAxisPar[AxisX1_NO].arrTargetPoint[3]:=arrAxisPar[AxisX1_NO].arrTargetPoint[1]+(103.94*COS(DEG_TO_RAD(-1+225))-103.94*COS(DEG_TO_RAD(225))); 
			arrAxisPar[AxisX2_NO].arrTargetPoint[3]:=arrAxisPar[AxisX2_NO].arrTargetPoint[1]+(103.94*SIN(DEG_TO_RAD(-1+315))-103.94*COS(DEG_TO_RAD(315)));
			arrAxisPar[AxisY_NO].arrTargetPoint[3]:=arrAxisPar[AxisY_NO].arrTargetPoint[1]+(103.94*COS(DEG_TO_RAD(-1+135))-103.94*COS(DEG_TO_RAD(135)));	
		iTest:=50;											
13:
		arrAxisPar[AxisX1_NO].arrTargetPoint[3]:=arrAxisPar[AxisX1_NO].arrTargetPoint[1]+(103.94*COS(DEG_TO_RAD(-2+225))-103.94*COS(DEG_TO_RAD(225))); 
			arrAxisPar[AxisX2_NO].arrTargetPoint[3]:=arrAxisPar[AxisX2_NO].arrTargetPoint[1]+(103.94*SIN(DEG_TO_RAD(-2+315))-103.94*COS(DEG_TO_RAD(315)));
			arrAxisPar[AxisY_NO].arrTargetPoint[3]:=arrAxisPar[AxisY_NO].arrTargetPoint[1]+(103.94*COS(DEG_TO_RAD(-2+135))-103.94*COS(DEG_TO_RAD(135)));	
		iTest:=50;							
14:
		arrAxisPar[AxisX1_NO].arrTargetPoint[3]:=arrAxisPar[AxisX1_NO].arrTargetPoint[1];//+(103.94*COS(DEG_TO_RAD(CCD_W+225))-103.94*COS(DEG_TO_RAD(225))); 
			arrAxisPar[AxisX2_NO].arrTargetPoint[3]:=arrAxisPar[AxisX2_NO].arrTargetPoint[1];//+(103.94*SIN(DEG_TO_RAD(CCD_W+315))-103.94*COS(DEG_TO_RAD(315)));
		arrAxisPar[AxisY_NO].arrTargetPoint[3]:=arrAxisPar[AxisY_NO].arrTargetPoint[1];//+(103.94*COS(DEG_TO_RAD(CCD_W+135))-103.94*COS(DEG_TO_RAD(135)));		
		iTest:=50;			
   
  50:  //先移动X1,X2
		
									  IF arrAxisCtrl[AxisX1_NO].Status.Homed AND arrAxisCtrl[AxisX1_NO].Status.NoMoving THEN
													IF arrAxisCtrl[AxisX1_NO].Cmd.arrbRealPoint[3] THEN
														arrAxisCtrl[AxisX1_NO].Cmd.iGoSetPos:=0;
													ELSE
														arrAxisCtrl[AxisX1_NO].Cmd.iGoSetPos:=3;
													END_IF
										END_IF
										IF arrAxisCtrl[AxisX2_NO].Status.Homed AND arrAxisCtrl[AxisX2_NO].Status.NoMoving  THEN
													IF arrAxisCtrl[AxisX2_NO].Cmd.arrbRealPoint[3] THEN
														arrAxisCtrl[AxisX2_NO].Cmd.iGoSetPos:=0;
													ELSE
														arrAxisCtrl[AxisX2_NO].Cmd.iGoSetPos:=3;
													END_IF
										END_IF	
										IF  arrAxisCtrl[AxisX1_NO].Cmd.arrbRealPoint[3]  AND arrAxisCtrl[AxisX1_NO].Status.NoMoving AND 
							 				arrAxisCtrl[AxisX2_NO].Cmd.arrbRealPoint[3] AND arrAxisCtrl[AxisX2_NO].Status.NoMoving THEN
											iTest:=60;		
										END_IF	
				
	60://再移动Y
		
									IF arrAxisCtrl[AxisY_NO].Status.Homed AND arrAxisCtrl[AxisY_NO].Status.NoMoving  THEN
												IF arrAxisCtrl[AxisY_NO].Cmd.arrbRealPoint[3] THEN
													arrAxisCtrl[AxisY_NO].Cmd.iGoSetPos:=0;
									                  bTest1:=FALSE;
														iTest:=66;									
												ELSE
													arrAxisCtrl[AxisY_NO].Cmd.iGoSetPos:=3;
												END_IF
									
								END_IF
	
		
END_CASE

END_IF

END_FUNCTION_BLOCK

// ---- P2POUs/BasicFunction/12_User2/FB_RecdevPla.TcPOU
FUNCTION_BLOCK FB_RecdevPla//正、负极片纠偏平台自动功能块
VAR_IN_OUT
	Step0: INT;//程序步
	RecdevStart:BOOL;//启动条件	
	RecdevDone:BOOL;//纠偏完成
END_VAR
VAR_INPUT
	RecdevAgree:BOOL;//纠偏允许
	AxisX1_NO : INT; //X1轴号
	AxisX2_NO : INT;//X2轴号
	AxisY_NO  : INT;//Y轴号
	CCD_X1:REAL;//CCD拍照X轴方向的纠偏值
	CCD_X2:REAL;//CCD拍照Y轴方的纠偏值
	CCD_Y:REAL;//CCD拍照旋转方向的纠偏值	
END_VAR

VAR_OUTPUT
END_VAR
VAR

END_VAR




//极片纠偏自动功能
CASE Step0 of
		0://等待纠偏启动
			IF RecdevStart THEN
				Step0:=10;
			END_IF
		10://根据CCD计算纠偏位移
			arrAxisPar[AxisX1_NO].arrTargetPoint[2]:=arrAxisPar[AxisX1_NO].arrTargetPoint[1]+CCD_X1;//+(103.94*COS(DEG_TO_RAD(CCD_W+225))-103.94*COS(DEG_TO_RAD(225))); 
			arrAxisPar[AxisX2_NO].arrTargetPoint[2]:=arrAxisPar[AxisX2_NO].arrTargetPoint[1]+CCD_X2;//+(103.94*SIN(DEG_TO_RAD(CCD_W+315))-103.94*COS(DEG_TO_RAD(315)));
			arrAxisPar[AxisY_NO].arrTargetPoint[2]:=arrAxisPar[AxisY_NO].arrTargetPoint[1]+CCD_Y;//+(103.94*COS(DEG_TO_RAD(CCD_W+135))-103.94*COS(DEG_TO_RAD(135)));	
			Step0:=20;	
		20://启动极片纠偏
		IF RecdevAgree THEN
				IF arrAxisCtrl[AxisX1_NO].Status.Homed AND arrAxisCtrl[AxisX1_NO].Status.NoMoving AND NOT arrAxisCtrl[AxisX1_NO].Status.Error THEN
							IF arrAxisCtrl[AxisX1_NO].Cmd.arrbRealPoint[2] THEN
								arrAxisCtrl[AxisX1_NO].Cmd.iGoSetPos:=0;
							ELSE
								arrAxisCtrl[AxisX1_NO].Cmd.iGoSetPos:=2;
							END_IF
				END_IF
				IF arrAxisCtrl[AxisX2_NO].Status.Homed AND arrAxisCtrl[AxisX2_NO].Status.NoMoving AND NOT arrAxisCtrl[AxisX2_NO].Status.Error THEN
							IF arrAxisCtrl[AxisX2_NO].Cmd.arrbRealPoint[2] THEN
								arrAxisCtrl[AxisX2_NO].Cmd.iGoSetPos:=0;
							ELSE
								arrAxisCtrl[AxisX2_NO].Cmd.iGoSetPos:=2;
							END_IF
				END_IF	
				IF arrAxisCtrl[AxisY_NO].Status.Homed AND arrAxisCtrl[AxisY_NO].Status.NoMoving AND NOT arrAxisCtrl[AxisY_NO].Status.Error THEN
							IF arrAxisCtrl[AxisY_NO].Cmd.arrbRealPoint[2] THEN
								arrAxisCtrl[AxisY_NO].Cmd.iGoSetPos:=0;
							ELSE
								arrAxisCtrl[AxisY_NO].Cmd.iGoSetPos:=2;
							END_IF
				END_IF
				IF  arrAxisCtrl[AxisX1_NO].Cmd.arrbRealPoint[2]  AND 	arrAxisCtrl[AxisX2_NO].Cmd.arrbRealPoint[2] AND  arrAxisCtrl[AxisY_NO].Cmd.arrbRealPoint[2] THEN
					RecdevDone:=TRUE;//置位纠偏完成
					RecdevStart:=FALSE;//复纠偏启动
					Step0:=0;
				END_IF	
		END_IF		
END_CASE

END_FUNCTION_BLOCK

// ---- P2POUs/BasicFunction/09_User1/FB_CrectCamMove.TcPOU
FUNCTION_BLOCK FB_CrectCamMove	
VAR_INPUT
   	bCreatTable		                         :BOOL;	
	Reset                                        :BOOL;  
	iTable		                            :UINT;    

    fMoveLength                             :REAL;   
    fMasterKeyPos                         :REAL;   
END_VAR

VAR_IN_OUT
	axisSlave		                            :axis_ref;  
	axisMaster		                            :axis_ref;  
END_VAR

VAR_OUTPUT
    bCreatTableDone                        :BOOL;
    bCreatTableError                        :BOOL;
	bError                         :BOOL;

END_VAR


VAR
	rtrigs		                                      :ARRAY[1..3]OF R_TRIG;
	ftrigs		                                      :ARRAY[1..3]OF F_TRIG;
    PositionData1			                  :ARRAY[1..4] OF MC_MotionFunctionPoint;	////
	fbCamtableselect:		               	MC_CamTableSelect;////
	Cam_table:				MC_CAM_REF;////
	bWriteCamData: BOOL;
    iCreatTableStep       :INT;
END_VAR


rtrigs[1](CLK:=bCreatTable);  
ftrigs[1](CLK:=bCreatTable);  

CASE iCreatTableStep OF   
0:  
    IF  rtrigs[1].Q  AND NOT bCreatTableError  THEN
         fbCamtableselect.Execute:=FALSE;
         bCreatTableDone:=FALSE;
         bCreatTable:=FALSE;
         bWriteCamData:=TRUE;
         iCreatTableStep:=10;
    END_IF 

10: 
   IF NOT bWriteCamData THEN 
	  fbCamtableselect.Execute:=TRUE;   
	 iCreatTableStep:=20;	
  END_IF

20:		
	IF NOT  fbCamtableselect.Execute   THEN
        bCreatTableDone:=TRUE;
		iCreatTableStep:=0;	
    ELSIF  fbCamtableselect.Error        THEN
       bCreatTableError:=TRUE;
       iCreatTableStep:=999;	//创建凸轮失败
	END_IF		
END_CASE

(**********故障***********)
	IF  Reset  AND bCreatTableError  THEN  
	   bCreatTableError:=FALSE;
	   iCreatTableStep:=0;
	END_IF


ModifyCam();

ACTION ModifyCam:

fbCamtableselect(   
	Execute:=                        fbCamtableselect.Execute ,
	Periodic:=                        FALSE ,
	MasterAbsolute:=             FALSE,
	SlaveAbsolute:=                FALSE ,
	CamTableID:=                  iTable,
	Master:=                         axisMaster ,
	Slave:=                            axisSlave ,
	CamTable:=                     Cam_table , );

IF fbCamtableselect.Done THEN
    fbCamtableselect.Execute:=FALSE;
END_IF

IF bWriteCamData  THEN
 
	  Cam_table.ArraySize:=SIZEOF(PositionData1); 
	  Cam_table.NoOfColumns:=1;
	  Cam_table.NoOfRows:=3;
	  Cam_table.pArray:=ADR(PositionData1);
	  Cam_table.TableType:=MC_TABLETYPE_MOTIONFUNCTION;
  
	  PositionData1[1].	PointIndex	:=	        1;
	  PositionData1[1].	FunctionType	:=		MOTIONFUNCTYPE_BESCHLTRAPEZ;//MOTIONFUNCTYPE_BESCHLTRAPEZ     MOTIONFUNCTYPE_POLYNOM7_MM    MOTIONFUNCTYPE_BESCHLTRAPEZ
	  PositionData1[1].	PointType	:=	        MOTIONPOINTTYPE_MOTION;
	  PositionData1[1].	RelIndexNextPoint	:=  1;
	  PositionData1[1].	MasterPos	:=	        0;
	  PositionData1[1].	SlavePos	:=	        0;		//fMoveLength
	  PositionData1[1].	SlaveVelo	:=	        0;
	  
	  PositionData1[2].	PointIndex	:=	        2;
	  PositionData1[2].	FunctionType	:=		MOTIONFUNCTYPE_POLYNOM1;
	  PositionData1[2].	PointType	:=	        MOTIONPOINTTYPE_MOTION;
	  PositionData1[2].	RelIndexNextPoint	:=  1;
	  PositionData1[2].	MasterPos	:=	        fMasterKeyPos;//fMasterKeyPos
	  PositionData1[2].	SlavePos	:=	        fMoveLength;	
	  PositionData1[2].	SlaveVelo	:=	        0	;

	  PositionData1[3].	PointIndex	:=	        3;
	  PositionData1[3].	FunctionType	:=		MOTIONFUNCTYPE_BESCHLTRAPEZ;
	  PositionData1[3].	PointType	:=	        MOTIONPOINTTYPE_MOTION;
	  PositionData1[3].	RelIndexNextPoint	:=  0;
	  PositionData1[3].	MasterPos	:=	        360;
	  PositionData1[3].	SlavePos	:=	        fMoveLength;	
	  PositionData1[3].	SlaveVelo	:=	        0	;

     bWriteCamData:=FALSE;
END_IF
END_ACTION

END_FUNCTION_BLOCK

// ---- P2POUs/BasicFunction/09_User1/FB_CrectCamUpDown.TcPOU
FUNCTION_BLOCK FB_CrectCamUpDown	
VAR_INPUT
   	bCreatTable		                         :BOOL;	
	Reset                                        :BOOL;  
	iTable		                                :UINT;    

	fInitLength									:REAL;//耦合的初始高度
    fMoveLength                              :REAL;   //目标取或放料高度
    fSaveLength                               :REAL;    //升降安全高度

    fMasterKeyPos1                           :REAL:=208;   
    fMasterKeyPos2                           :REAL:=256;   
    fMasterKeyPos3                           :REAL:=328;   
	fMasterKeyPos4                           :REAL:=328;   
	fMasterKeyPos5                           :REAL;   
	fMasterKeyPos6                           :REAL;   
	
	fSlaveVelo                                    :REAL:=0.32;  
	
END_VAR

VAR_IN_OUT
	axisSlave		                            :axis_ref;  
	axisMaster		                            :axis_ref;  
END_VAR

VAR_OUTPUT
    bCreatTableDone                        :BOOL;
    bCreatTableError                        :BOOL;
	bError                         :BOOL;

END_VAR


VAR
	rtrigs		                                      :ARRAY[1..3]OF R_TRIG;
	ftrigs		                                      :ARRAY[1..3]OF F_TRIG;
    PositionData1			                  :ARRAY[1..8] OF MC_MotionFunctionPoint;	////
	fbCamtableselect:		               	MC_CamTableSelect;////
	Cam_table:				MC_CAM_REF;////
	bWriteCamData: BOOL;
    iCreatTableStep       :INT;
END_VAR


rtrigs[1](CLK:=bCreatTable);  
ftrigs[1](CLK:=bCreatTable);  

CASE iCreatTableStep OF   
0:  
    IF  rtrigs[1].Q  AND NOT bCreatTableError  THEN
         fbCamtableselect.Execute:=FALSE;
         bCreatTableDone:=FALSE;
         bCreatTable:=FALSE;
         bWriteCamData:=TRUE;
         iCreatTableStep:=10;
    END_IF 

10: 
   IF NOT bWriteCamData THEN 
	  fbCamtableselect.Execute:=TRUE;   
	 iCreatTableStep:=20;	
  END_IF

20:		
	IF NOT  fbCamtableselect.Execute   THEN
        bCreatTableDone:=TRUE;
		iCreatTableStep:=0;	
    ELSIF  fbCamtableselect.Error        THEN
       bCreatTableError:=TRUE;
       iCreatTableStep:=999;	//创建凸轮失败
	END_IF		
END_CASE

(**********故障***********)
	IF  Reset  AND bCreatTableError  THEN  
	   bCreatTableError:=FALSE;
	   iCreatTableStep:=0;
	END_IF


ModifyCam();

ACTION ModifyCam:

fbCamtableselect(   
	Execute:=                        fbCamtableselect.Execute ,
	Periodic:=                        FALSE ,
	MasterAbsolute:=             FALSE,
	SlaveAbsolute:=                FALSE ,
	CamTableID:=                  iTable,
	Master:=                         axisMaster ,
	Slave:=                            axisSlave ,
	CamTable:=                     Cam_table , );

IF fbCamtableselect.Done THEN
    fbCamtableselect.Execute:=FALSE;
END_IF


IF bWriteCamData  THEN
	  Cam_table.ArraySize:=SIZEOF(PositionData1); 
	  Cam_table.NoOfColumns:=1;
	  Cam_table.NoOfRows:=4;
	  Cam_table.pArray:=ADR(PositionData1);
	  Cam_table.TableType:=MC_TABLETYPE_MOTIONFUNCTION;
  
      //MOTIONFUNCTYPE_BESCHLTRAPEZ     MOTIONFUNCTYPE_POLYNOM7_MM    MOTIONFUNCTYPE_BESCHLTRAPEZ   MOTIONFUNCTYPE_POLYNOM1
	  PositionData1[1].	PointIndex	:=	        1;
	  PositionData1[1].	FunctionType	:=		MOTIONFUNCTYPE_POLYNOM5_MM;//MOTIONFUNCTYPE_BESCHLTRAPEZ     MOTIONFUNCTYPE_POLYNOM7_MM    MOTIONFUNCTYPE_BESCHLTRAPEZ
	  PositionData1[1].	PointType	:=	        MOTIONPOINTTYPE_MOTION;
	  PositionData1[1].	RelIndexNextPoint	:=  1;
	  PositionData1[1].	MasterPos	:=	        0;
	  PositionData1[1].	SlavePos	:=	        0;		//fMoveLength
	  PositionData1[1].	SlaveVelo	:=	        0;
	  
	  PositionData1[2].	PointIndex	:=	        2;
	  PositionData1[2].	FunctionType	:=		MOTIONFUNCTYPE_POLYNOM5_MM;
	  PositionData1[2].	PointType	:=	        MOTIONPOINTTYPE_MOTION;
	  PositionData1[2].	RelIndexNextPoint	:=  1;
	  PositionData1[2].	MasterPos	:=	        fMasterKeyPos1;//fMasterKeyPos
	  PositionData1[2].	SlavePos	:=	        fSaveLength ;	
	  PositionData1[2].	SlaveVelo	:=	        0;//(fInitLength-fSaveLength)/fMasterKeyPos1	;
	  
	  PositionData1[3].	PointIndex	:=	        3;
	  PositionData1[3].	FunctionType	:=		MOTIONFUNCTYPE_POLYNOM1;
	  PositionData1[3].	PointType	:=	        MOTIONPOINTTYPE_MOTION;
	  PositionData1[3].	RelIndexNextPoint	:=  1;
	  PositionData1[3].	MasterPos	:=	        fMasterKeyPos2;//fMasterKeyPos
	  PositionData1[3].	SlavePos	:=	        fMoveLength;	
	  PositionData1[3].	SlaveVelo	:=	        0;//(fInitLength-fSaveLength)/fMasterKeyPos1	;  
	  
	  PositionData1[4].	PointIndex	:=	        4;
	  PositionData1[4].	FunctionType	:=		MOTIONFUNCTYPE_POLYNOM5_MM;
	  PositionData1[4].	PointType	:=	        MOTIONPOINTTYPE_MOTION;
	  PositionData1[4].	RelIndexNextPoint	:=  0;
	  PositionData1[4].	MasterPos	:=	        360;
	  PositionData1[4].	SlavePos	:=	        fMoveLength;	
	  PositionData1[4].	SlaveVelo	:=	        0	;
     bWriteCamData:=FALSE;
END_IF













(*
IF bWriteCamData  THEN
 
	  Cam_table.ArraySize:=SIZEOF(PositionData1); 
	  Cam_table.NoOfColumns:=1;
	  Cam_table.NoOfRows:=7;
	  Cam_table.pArray:=ADR(PositionData1);
	  Cam_table.TableType:=MC_TABLETYPE_MOTIONFUNCTION;
  
      //MOTIONFUNCTYPE_BESCHLTRAPEZ     MOTIONFUNCTYPE_POLYNOM7_MM    MOTIONFUNCTYPE_BESCHLTRAPEZ   MOTIONFUNCTYPE_POLYNOM1

	  PositionData1[1].	PointIndex	:=	        1;
	  PositionData1[1].	FunctionType	:=		MOTIONFUNCTYPE_POLYNOM5_MM;//MOTIONFUNCTYPE_BESCHLTRAPEZ     MOTIONFUNCTYPE_POLYNOM7_MM    MOTIONFUNCTYPE_BESCHLTRAPEZ
	  PositionData1[1].	PointType	:=	        MOTIONPOINTTYPE_MOTION;
	  PositionData1[1].	RelIndexNextPoint	:=  1;
	  PositionData1[1].	MasterPos	:=	        0;
	  PositionData1[1].	SlavePos	:=	        0;		//fMoveLength
	  PositionData1[1].	SlaveVelo	:=	        0;
	  
	  PositionData1[2].	PointIndex	:=	        2;
	  PositionData1[2].	FunctionType	:=		MOTIONFUNCTYPE_POLYNOM5_MM;
	  PositionData1[2].	PointType	:=	        MOTIONPOINTTYPE_MOTION;
	  PositionData1[2].	RelIndexNextPoint	:=  1;
	  PositionData1[2].	MasterPos	:=	        fMasterKeyPos1;//fMasterKeyPos
	  PositionData1[2].	SlavePos	:=	        fSaveLength - fInitLength;	
	  PositionData1[2].	SlaveVelo	:=	        0;//(fInitLength-fSaveLength)/fMasterKeyPos1	;

	  PositionData1[3].	PointIndex	:=	        3;//SJ
	  PositionData1[3].	FunctionType	:=		MOTIONFUNCTYPE_POLYNOM1;
	  PositionData1[3].	PointType	:=	        MOTIONPOINTTYPE_MOTION;
	  PositionData1[3].	RelIndexNextPoint	:=  1;
	  PositionData1[3].	MasterPos	:=	        fMasterKeyPos2-10;//fMasterKeyPos
	  PositionData1[3].	SlavePos	:=	        0;	
	  PositionData1[3].	SlaveVelo	:=	        0;//(fInitLength-fSaveLength)/fMasterKeyPos1	;	  
	  
	  
	  PositionData1[4].	PointIndex	:=	        4;
	  PositionData1[4].	FunctionType	:=		MOTIONFUNCTYPE_POLYNOM5_MM;
	  PositionData1[4].	PointType	:=	        MOTIONPOINTTYPE_MOTION;
	  PositionData1[4].	RelIndexNextPoint	:=  1;
	  PositionData1[4].	MasterPos	:=	        fMasterKeyPos2;//fMasterKeyPos
	  PositionData1[4].	SlavePos	:=	        0;	
	  PositionData1[4].	SlaveVelo	:=	        0;//(fInitLength-fSaveLength)/fMasterKeyPos1	;
	  
	  PositionData1[5].	PointIndex	:=	        5;
	  PositionData1[5].	FunctionType	:=		MOTIONFUNCTYPE_POLYNOM1;
	  PositionData1[5].	PointType	:=	        MOTIONPOINTTYPE_MOTION;
	  PositionData1[5].	RelIndexNextPoint	:=  1;
	  PositionData1[5].	MasterPos	:=	        fMasterKeyPos3;
	  PositionData1[5].	SlavePos	:=	        12;	//
	  PositionData1[5].	SlaveVelo	:=	        0	;

	  PositionData1[6].	PointIndex	:=	        6;
	  PositionData1[6].	FunctionType	:=		MOTIONFUNCTYPE_POLYNOM5_MM;
	  PositionData1[6].	PointType	:=	        MOTIONPOINTTYPE_MOTION;
	  PositionData1[6].	RelIndexNextPoint	:=  1;
	  PositionData1[6].	MasterPos	:=	        fMasterKeyPos4;//fMasterKeyPos
	  PositionData1[6].	SlavePos	:=	    12   ;	 // fMoveLength-fInitLength
	  PositionData1[6].	SlaveVelo	:=	       0	;

	  PositionData1[7].	PointIndex	:=	        7;
	  PositionData1[7].	FunctionType	:=		MOTIONFUNCTYPE_POLYNOM5_MM;
	  PositionData1[7].	PointType	:=	        MOTIONPOINTTYPE_MOTION;
	  PositionData1[7].	RelIndexNextPoint	:=  0;
	  PositionData1[7].	MasterPos	:=	        360;
	  PositionData1[7].	SlavePos	:=	        12;	
	  PositionData1[7].	SlaveVelo	:=	       0	;


     bWriteCamData:=FALSE;
END_IF

*)
END_ACTION

END_FUNCTION_BLOCK

// ---- P2POUs/BasicFunction/09_User1/FB_CrectCamUpDown_1.TcPOU
FUNCTION_BLOCK FB_CrectCamUpDown_1	
VAR_INPUT
   	bCreatTable		                         :BOOL;	
	Reset                                        :BOOL;  
	iTable		                                :UINT;    

	fInitLength									:REAL;//耦合的初始高度
    fMoveLength                              :REAL;   //目标取或放料高度
    fSaveLength                               :REAL;    //升降安全高度

    fMasterKeyPos1                           :REAL:=72;   
    fMasterKeyPos2                           :REAL:=144;   
    fMasterKeyPos3                           :REAL:=261;   
	fMasterKeyPos4                           :REAL:=297;   
	fMasterKeyPos5                           :REAL:=328;   	
	fMasterKeyPos6                           :REAL:=328;   	
	fSlaveVelo                                    :REAL:=0.32;   	  
	
END_VAR

VAR_IN_OUT
	axisSlave		                            :axis_ref;  
	axisMaster		                            :axis_ref;  
END_VAR

VAR_OUTPUT
    bCreatTableDone                        :BOOL;
    bCreatTableError                        :BOOL;
	bError                         :BOOL;

END_VAR


VAR
	rtrigs		                                      :ARRAY[1..3]OF R_TRIG;
	ftrigs		                                      :ARRAY[1..3]OF F_TRIG;
    PositionData1			                  :ARRAY[1..8] OF MC_MotionFunctionPoint;	////
	fbCamtableselect:		               	MC_CamTableSelect;////
	Cam_table:				MC_CAM_REF;////
	bWriteCamData: BOOL;
    iCreatTableStep       :INT;
END_VAR


rtrigs[1](CLK:=bCreatTable);  
ftrigs[1](CLK:=bCreatTable);  

CASE iCreatTableStep OF   
0:  
    IF  rtrigs[1].Q  AND NOT bCreatTableError  THEN
         fbCamtableselect.Execute:=FALSE;
         bCreatTableDone:=FALSE;
         bCreatTable:=FALSE;
         bWriteCamData:=TRUE;
         iCreatTableStep:=10;
    END_IF 

10: 
   IF NOT bWriteCamData THEN 
	  fbCamtableselect.Execute:=TRUE;   
	 iCreatTableStep:=20;	
  END_IF

20:		
	IF NOT  fbCamtableselect.Execute   THEN
        bCreatTableDone:=TRUE;
		iCreatTableStep:=0;	
    ELSIF  fbCamtableselect.Error        THEN
       bCreatTableError:=TRUE;
       iCreatTableStep:=999;	//创建凸轮失败
	END_IF		
END_CASE

(**********故障***********)
	IF  Reset  AND bCreatTableError  THEN  
	   bCreatTableError:=FALSE;
	   iCreatTableStep:=0;
	END_IF


ModifyCam();

ACTION ModifyCam:

fbCamtableselect(   
	Execute:=                        fbCamtableselect.Execute ,
	Periodic:=                        FALSE ,
	MasterAbsolute:=             FALSE,
	SlaveAbsolute:=                FALSE ,
	CamTableID:=                  iTable,
	Master:=                         axisMaster ,
	Slave:=                            axisSlave ,
	CamTable:=                     Cam_table , );

IF fbCamtableselect.Done THEN
    fbCamtableselect.Execute:=FALSE;
END_IF

IF bWriteCamData  THEN
 
	  Cam_table.ArraySize:=SIZEOF(PositionData1); 
	  Cam_table.NoOfColumns:=1;
	  Cam_table.NoOfRows:=7;
	  Cam_table.pArray:=ADR(PositionData1);
	  Cam_table.TableType:=MC_TABLETYPE_MOTIONFUNCTION;
  
      //MOTIONFUNCTYPE_BESCHLTRAPEZ     MOTIONFUNCTYPE_POLYNOM7_MM    MOTIONFUNCTYPE_BESCHLTRAPEZ   MOTIONFUNCTYPE_POLYNOM1

	  PositionData1[1].	PointIndex	:=	        1;
	  PositionData1[1].	FunctionType	:=		MOTIONFUNCTYPE_POLYNOM5_MM;//MOTIONFUNCTYPE_BESCHLTRAPEZ     MOTIONFUNCTYPE_POLYNOM7_MM    MOTIONFUNCTYPE_BESCHLTRAPEZ
	  PositionData1[1].	PointType	:=	        MOTIONPOINTTYPE_MOTION;
	  PositionData1[1].	RelIndexNextPoint	:=  1;
	  PositionData1[1].	MasterPos	:=	        0;
	  PositionData1[1].	SlavePos	:=	        0;		//fMoveLength
	  PositionData1[1].	SlaveVelo	:=	        0;
	  
	  PositionData1[2].	PointIndex	:=	        2;
	  PositionData1[2].	FunctionType	:=		MOTIONFUNCTYPE_POLYNOM5_MM;
	  PositionData1[2].	PointType	:=	        MOTIONPOINTTYPE_MOTION;
	  PositionData1[2].	RelIndexNextPoint	:=  1;
	  PositionData1[2].	MasterPos	:=	        fMasterKeyPos1;//fMasterKeyPos
	  PositionData1[2].	SlavePos	:=	        fSaveLength ;	
	  PositionData1[2].	SlaveVelo	:=	        0;//(fInitLength-fSaveLength)/fMasterKeyPos1	;
	  
	  PositionData1[3].	PointIndex	:=	        3;
	  PositionData1[3].	FunctionType	:=		MOTIONFUNCTYPE_POLYNOM5_MM;
	  PositionData1[3].	PointType	:=	        MOTIONPOINTTYPE_MOTION;
	  PositionData1[3].	RelIndexNextPoint	:=  1;
	  PositionData1[3].	MasterPos	:=	        fMasterKeyPos2;//fMasterKeyPos
	  PositionData1[3].	SlavePos	:=	        fMoveLength-4;	
	  PositionData1[3].	SlaveVelo	:=	        fSlaveVelo;//(fInitLength-fSaveLength)/fMasterKeyPos1	;  
	  
	  PositionData1[4].	PointIndex	:=	        4;
	  PositionData1[4].	FunctionType	:=		MOTIONFUNCTYPE_POLYNOM1;
	  PositionData1[4].	PointType	:=	        MOTIONPOINTTYPE_MOTION;
	  PositionData1[4].	RelIndexNextPoint	:=  1;
	  PositionData1[4].	MasterPos	:=	        fMasterKeyPos3;
	  PositionData1[4].	SlavePos	:=	        fMoveLength;	
	  PositionData1[4].	SlaveVelo	:=	        0	;

	  PositionData1[5].	PointIndex	:=	        5;
	  PositionData1[5].	FunctionType	:=		MOTIONFUNCTYPE_POLYNOM5_MM;
	  PositionData1[5].	PointType	:=	        MOTIONPOINTTYPE_MOTION;
	  PositionData1[5].	RelIndexNextPoint	:=  1;
	  PositionData1[5].	MasterPos	:=	        fMasterKeyPos4;//fMasterKeyPos
	  PositionData1[5].	SlavePos	:=	        fMoveLength;	
	  PositionData1[5].	SlaveVelo	:=	       0	;

	  PositionData1[6].	PointIndex	:=	        6;
	  PositionData1[6].	FunctionType	:=		MOTIONFUNCTYPE_POLYNOM5_MM;
	  PositionData1[6].	PointType	:=	        MOTIONPOINTTYPE_MOTION;
	  PositionData1[6].	RelIndexNextPoint	:=  1;
	  PositionData1[6].	MasterPos	:=	        fMasterKeyPos5;
	  PositionData1[6].	SlavePos	:=	        0;	
	  PositionData1[6].	SlaveVelo	:=	       0	;

	  PositionData1[7].	PointIndex	:=	        7;
	  PositionData1[7].	FunctionType	:=		MOTIONFUNCTYPE_POLYNOM5_MM;
	  PositionData1[7].	PointType	:=	        MOTIONPOINTTYPE_MOTION;
	  PositionData1[7].	RelIndexNextPoint	:=  0;
	  PositionData1[7].	MasterPos	:=	        360;
	  PositionData1[7].	SlavePos	:=	        0;	
	  PositionData1[7].	SlaveVelo	:=	       0	;

     bWriteCamData:=FALSE;
END_IF




(*

IF bWriteCamData  THEN
 
	  Cam_table.ArraySize:=SIZEOF(PositionData1); 
	  Cam_table.NoOfColumns:=1;
	  Cam_table.NoOfRows:=8;
	  Cam_table.pArray:=ADR(PositionData1);
	  Cam_table.TableType:=MC_TABLETYPE_MOTIONFUNCTION;
  
      //MOTIONFUNCTYPE_BESCHLTRAPEZ     MOTIONFUNCTYPE_POLYNOM7_MM    MOTIONFUNCTYPE_BESCHLTRAPEZ   MOTIONFUNCTYPE_POLYNOM1

	  PositionData1[1].	PointIndex	:=	        1;
	  PositionData1[1].	FunctionType	:=		MOTIONFUNCTYPE_POLYNOM5_MM;//MOTIONFUNCTYPE_BESCHLTRAPEZ     MOTIONFUNCTYPE_POLYNOM7_MM    MOTIONFUNCTYPE_BESCHLTRAPEZ
	  PositionData1[1].	PointType	:=	        MOTIONPOINTTYPE_MOTION;
	  PositionData1[1].	RelIndexNextPoint	:=  1;
	  PositionData1[1].	MasterPos	:=	        0;
	  PositionData1[1].	SlavePos	:=	        0;		//fMoveLength
	  PositionData1[1].	SlaveVelo	:=	        0;
	  
	  PositionData1[2].	PointIndex	:=	        2;
	  PositionData1[2].	FunctionType	:=		MOTIONFUNCTYPE_POLYNOM5_MM;
	  PositionData1[2].	PointType	:=	        MOTIONPOINTTYPE_MOTION;
	  PositionData1[2].	RelIndexNextPoint	:=  1;
	  PositionData1[2].	MasterPos	:=	        fMasterKeyPos1;//fMasterKeyPos
	  PositionData1[2].	SlavePos	:=	        fSaveLength - fInitLength;	
	  PositionData1[2].	SlaveVelo	:=	        0;//(fInitLength-fSaveLength)/fMasterKeyPos1	;

	  PositionData1[3].	PointIndex	:=	        3;
	  PositionData1[3].	FunctionType	:=		MOTIONFUNCTYPE_POLYNOM5_MM;
	  PositionData1[3].	PointType	:=	        MOTIONPOINTTYPE_MOTION;
	  PositionData1[3].	RelIndexNextPoint	:=  1;
	  PositionData1[3].	MasterPos	:=	        fMasterKeyPos2;//fMasterKeyPos
	  PositionData1[3].	SlavePos	:=	        0;	
	  PositionData1[3].	SlaveVelo	:=	        0;//(fInitLength-fSaveLength)/fMasterKeyPos1	;
	  
	  PositionData1[4].	PointIndex	:=	        4;
	  PositionData1[4].	FunctionType	:=		MOTIONFUNCTYPE_POLYNOM5_MM;
	  PositionData1[4].	PointType	:=	        MOTIONPOINTTYPE_MOTION;
	  PositionData1[4].	RelIndexNextPoint	:=  1;
	  PositionData1[4].	MasterPos	:=	        fMasterKeyPos6;//fMasterKeyPos
	  PositionData1[4].	SlavePos	:=	        fMoveLength-fInitLength-4;	
	  PositionData1[4].	SlaveVelo	:=	        fSlaveVelo;//(fInitLength-fSaveLength)/fMasterKeyPos1	;  
	  
	  PositionData1[5].	PointIndex	:=	        5;
	  PositionData1[5].	FunctionType	:=		MOTIONFUNCTYPE_POLYNOM1;
	  PositionData1[5].	PointType	:=	        MOTIONPOINTTYPE_MOTION;
	  PositionData1[5].	RelIndexNextPoint	:=  1;
	  PositionData1[5].	MasterPos	:=	        fMasterKeyPos3;
	  PositionData1[5].	SlavePos	:=	        fMoveLength-fInitLength;	
	  PositionData1[5].	SlaveVelo	:=	        0	;

	  PositionData1[6].	PointIndex	:=	        6;
	  PositionData1[6].	FunctionType	:=		MOTIONFUNCTYPE_POLYNOM5_MM;
	  PositionData1[6].	PointType	:=	        MOTIONPOINTTYPE_MOTION;
	  PositionData1[6].	RelIndexNextPoint	:=  1;
	  PositionData1[6].	MasterPos	:=	        fMasterKeyPos4;//fMasterKeyPos
	  PositionData1[6].	SlavePos	:=	        fMoveLength-fInitLength;	
	  PositionData1[6].	SlaveVelo	:=	       0	;

	  PositionData1[7].	PointIndex	:=	        7;
	  PositionData1[7].	FunctionType	:=		MOTIONFUNCTYPE_POLYNOM5_MM;
	  PositionData1[7].	PointType	:=	        MOTIONPOINTTYPE_MOTION;
	  PositionData1[7].	RelIndexNextPoint	:=  1;
	  PositionData1[7].	MasterPos	:=	        fMasterKeyPos5;
	  PositionData1[7].	SlavePos	:=	        0;	
	  PositionData1[7].	SlaveVelo	:=	       0	;

	  PositionData1[8].	PointIndex	:=	        8;
	  PositionData1[8].	FunctionType	:=		MOTIONFUNCTYPE_POLYNOM5_MM;
	  PositionData1[8].	PointType	:=	        MOTIONPOINTTYPE_MOTION;
	  PositionData1[8].	RelIndexNextPoint	:=  0;
	  PositionData1[8].	MasterPos	:=	        360;
	  PositionData1[8].	SlavePos	:=	        0;	
	  PositionData1[8].	SlaveVelo	:=	       0	;

     bWriteCamData:=FALSE;
END_IF

*)
END_ACTION

END_FUNCTION_BLOCK

// ---- P2POUs/BasicFunction/09_User1/FB_CrectCamUpDown_10.TcPOU
FUNCTION_BLOCK FB_CrectCamUpDown_10	
VAR_INPUT
   	bCreatTable		                         :BOOL;	
	Reset                                        :BOOL;  
	iTable		                                :UINT;    

	fInitLength									:REAL;//耦合的初始高度
    fMoveLength                              :REAL;   //目标取或放料高度
    fSaveLength                               :REAL;    //升降安全高度

    fMasterKeyPos1                           :REAL:=72;   
    fMasterKeyPos2                           :REAL:=144;   
    fMasterKeyPos3                           :REAL:=261;   
	fMasterKeyPos4                           :REAL:=297;   
	fMasterKeyPos5                           :REAL:=328;   	
	fMasterKeyPos6                           :REAL:=328;   	
	fSlaveVelo                                    :REAL:=0.32;   	  
	
END_VAR

VAR_IN_OUT
	axisSlave		                            :axis_ref;  
	axisMaster		                            :axis_ref;  
END_VAR

VAR_OUTPUT
    bCreatTableDone                        :BOOL;
    bCreatTableError                        :BOOL;
	bError                         :BOOL;

END_VAR


VAR
	rtrigs		                                      :ARRAY[1..3]OF R_TRIG;
	ftrigs		                                      :ARRAY[1..3]OF F_TRIG;
    PositionData1			                  :ARRAY[1..8] OF MC_MotionFunctionPoint;	////
	fbCamtableselect:		               	MC_CamTableSelect;////
	Cam_table:				MC_CAM_REF;////
	bWriteCamData: BOOL;
    iCreatTableStep       :INT;
END_VAR


rtrigs[1](CLK:=bCreatTable);  
ftrigs[1](CLK:=bCreatTable);  

CASE iCreatTableStep OF   
0:  
    IF  rtrigs[1].Q  AND NOT bCreatTableError  THEN
         fbCamtableselect.Execute:=FALSE;
         bCreatTableDone:=FALSE;
         bCreatTable:=FALSE;
         bWriteCamData:=TRUE;
         iCreatTableStep:=10;
    END_IF 

10: 
   IF NOT bWriteCamData THEN 
	  fbCamtableselect.Execute:=TRUE;   
	 iCreatTableStep:=20;	
  END_IF

20:		
	IF NOT  fbCamtableselect.Execute   THEN
        bCreatTableDone:=TRUE;
		iCreatTableStep:=0;	
    ELSIF  fbCamtableselect.Error        THEN
       bCreatTableError:=TRUE;
       iCreatTableStep:=999;	//创建凸轮失败
	END_IF		
END_CASE

(**********故障***********)
	IF  Reset  AND bCreatTableError  THEN  
	   bCreatTableError:=FALSE;
	   iCreatTableStep:=0;
	END_IF


ModifyCam();

ACTION ModifyCam:

fbCamtableselect(   
	Execute:=                        fbCamtableselect.Execute ,
	Periodic:=                        FALSE ,
	MasterAbsolute:=             FALSE,
	SlaveAbsolute:=                FALSE ,
	CamTableID:=                  iTable,
	Master:=                         axisMaster ,
	Slave:=                            axisSlave ,
	CamTable:=                     Cam_table , );

IF fbCamtableselect.Done THEN
    fbCamtableselect.Execute:=FALSE;
END_IF


IF bWriteCamData  THEN
 
	  Cam_table.ArraySize:=SIZEOF(PositionData1); 
	  Cam_table.NoOfColumns:=1;
	  Cam_table.NoOfRows:=4;
	  Cam_table.pArray:=ADR(PositionData1);
	  Cam_table.TableType:=MC_TABLETYPE_MOTIONFUNCTION;
  
      //MOTIONFUNCTYPE_BESCHLTRAPEZ     MOTIONFUNCTYPE_POLYNOM7_MM    MOTIONFUNCTYPE_BESCHLTRAPEZ   MOTIONFUNCTYPE_POLYNOM1
	  PositionData1[1].	PointIndex	:=	        1;
	  PositionData1[1].	FunctionType	:=		MOTIONFUNCTYPE_POLYNOM5_MM;//MOTIONFUNCTYPE_BESCHLTRAPEZ     MOTIONFUNCTYPE_POLYNOM7_MM    MOTIONFUNCTYPE_BESCHLTRAPEZ
	  PositionData1[1].	PointType	:=	        MOTIONPOINTTYPE_MOTION;
	  PositionData1[1].	RelIndexNextPoint	:=  1;
	  PositionData1[1].	MasterPos	:=	        0;
	  PositionData1[1].	SlavePos	:=	        0;		//fMoveLength
	  PositionData1[1].	SlaveVelo	:=	        0;
	  
	  PositionData1[2].	PointIndex	:=	        2;
	  PositionData1[2].	FunctionType	:=		MOTIONFUNCTYPE_POLYNOM5_MM;
	  PositionData1[2].	PointType	:=	        MOTIONPOINTTYPE_MOTION;
	  PositionData1[2].	RelIndexNextPoint	:=  1;
	  PositionData1[2].	MasterPos	:=	        fMasterKeyPos1;//fMasterKeyPos
	  PositionData1[2].	SlavePos	:=	        fSaveLength ;	
	  PositionData1[2].	SlaveVelo	:=	        0;//(fInitLength-fSaveLength)/fMasterKeyPos1	;
	  
	  PositionData1[3].	PointIndex	:=	        3;
	  PositionData1[3].	FunctionType	:=		MOTIONFUNCTYPE_POLYNOM1;
	  PositionData1[3].	PointType	:=	        MOTIONPOINTTYPE_MOTION;
	  PositionData1[3].	RelIndexNextPoint	:=  1;
	  PositionData1[3].	MasterPos	:=	        fMasterKeyPos2;//fMasterKeyPos
	  PositionData1[3].	SlavePos	:=	        0;	
	  PositionData1[3].	SlaveVelo	:=	        0;//(fInitLength-fSaveLength)/fMasterKeyPos1	;  
	  
	  PositionData1[4].	PointIndex	:=	        4;
	  PositionData1[4].	FunctionType	:=		MOTIONFUNCTYPE_POLYNOM5_MM;
	  PositionData1[4].	PointType	:=	        MOTIONPOINTTYPE_MOTION;
	  PositionData1[4].	RelIndexNextPoint	:= 0;
	  PositionData1[4].	MasterPos	:=	        360;
	  PositionData1[4].	SlavePos	:=	        0;	
	  PositionData1[4].	SlaveVelo	:=	        0	;

     bWriteCamData:=FALSE;
END_IF
END_ACTION

END_FUNCTION_BLOCK

// ---- P2POUs/BasicFunction/09_User1/FB_CrectCamUpDown_3.TcPOU
FUNCTION_BLOCK FB_CrectCamUpDown_3	
VAR_INPUT
   	bCreatTable		                         :BOOL;	
	Reset                                        :BOOL;  
	iTable		                                :UINT;    

	fInitLength									:REAL;//耦合的初始高度
    fMoveLength                              :REAL;   //目标取或放料高度
    fSaveLength                               :REAL;    //升降安全高度

    fMasterKeyPos1                           :REAL:=72;   
    fMasterKeyPos2                           :REAL:=144;   
    fMasterKeyPos3                           :REAL:=225;   
	fMasterKeyPos4                           :REAL:=261;   
	fMasterKeyPos5                           :REAL:=297;   
	fMasterKeyPos6                           :REAL:=328;   	
    fSlaveVelo                                    :REAL:=0.32;   	  
	
END_VAR

VAR_IN_OUT
	axisSlave		                            :axis_ref;  
	axisMaster		                            :axis_ref;  
END_VAR

VAR_OUTPUT
    bCreatTableDone                        :BOOL;
    bCreatTableError                        :BOOL;
	bError                         :BOOL;

END_VAR


VAR
	rtrigs		                                      :ARRAY[1..3]OF R_TRIG;
	ftrigs		                                      :ARRAY[1..3]OF F_TRIG;
    PositionData1			                  :ARRAY[1..8] OF MC_MotionFunctionPoint;	////
	fbCamtableselect:		               	MC_CamTableSelect;////
	Cam_table:				MC_CAM_REF;////
	bWriteCamData: BOOL;
    iCreatTableStep       :INT;
END_VAR


rtrigs[1](CLK:=bCreatTable);  
ftrigs[1](CLK:=bCreatTable);  

CASE iCreatTableStep OF   
0:  
    IF  rtrigs[1].Q  AND NOT bCreatTableError  THEN
         fbCamtableselect.Execute:=FALSE;
         bCreatTableDone:=FALSE;
         bCreatTable:=FALSE;
         bWriteCamData:=TRUE;
         iCreatTableStep:=10;
    END_IF 

10: 
   IF NOT bWriteCamData THEN 
	  fbCamtableselect.Execute:=TRUE;   
	 iCreatTableStep:=20;	
  END_IF

20:		
	IF NOT  fbCamtableselect.Execute   THEN
        bCreatTableDone:=TRUE;
		iCreatTableStep:=0;	
    ELSIF  fbCamtableselect.Error        THEN
       bCreatTableError:=TRUE;
       iCreatTableStep:=999;	//创建凸轮失败
	END_IF		
END_CASE

(**********故障***********)
	IF  Reset  AND bCreatTableError  THEN  
	   bCreatTableError:=FALSE;
	   iCreatTableStep:=0;
	END_IF


ModifyCam();

ACTION ModifyCam:

fbCamtableselect(   
	Execute:=                        fbCamtableselect.Execute ,
	Periodic:=                        FALSE ,
	MasterAbsolute:=             FALSE,
	SlaveAbsolute:=                FALSE ,
	CamTableID:=                  iTable,
	Master:=                         axisMaster ,
	Slave:=                            axisSlave ,
	CamTable:=                     Cam_table , );

IF fbCamtableselect.Done THEN
    fbCamtableselect.Execute:=FALSE;
END_IF


IF bWriteCamData  THEN
	  Cam_table.ArraySize:=SIZEOF(PositionData1); 
	  Cam_table.NoOfColumns:=1;
	  Cam_table.NoOfRows:=7;
	  Cam_table.pArray:=ADR(PositionData1);
	  Cam_table.TableType:=MC_TABLETYPE_MOTIONFUNCTION;
  
      //MOTIONFUNCTYPE_BESCHLTRAPEZ     MOTIONFUNCTYPE_POLYNOM7_MM    MOTIONFUNCTYPE_BESCHLTRAPEZ   MOTIONFUNCTYPE_POLYNOM1

	  PositionData1[1].	PointIndex	:=	        1;
	  PositionData1[1].	FunctionType	:=		MOTIONFUNCTYPE_POLYNOM5_MM;//MOTIONFUNCTYPE_BESCHLTRAPEZ     MOTIONFUNCTYPE_POLYNOM7_MM    MOTIONFUNCTYPE_BESCHLTRAPEZ
	  PositionData1[1].	PointType	:=	        MOTIONPOINTTYPE_MOTION;
	  PositionData1[1].	RelIndexNextPoint	:=  1;
	  PositionData1[1].	MasterPos	:=	        0;
	  PositionData1[1].	SlavePos	:=	        0;		//fMoveLength
	  PositionData1[1].	SlaveVelo	:=	        0;
	  
	  PositionData1[2].	PointIndex	:=	        2;
	  PositionData1[2].	FunctionType	:=		MOTIONFUNCTYPE_POLYNOM5_MM;
	  PositionData1[2].	PointType	:=	        MOTIONPOINTTYPE_MOTION;
	  PositionData1[2].	RelIndexNextPoint	:=  1;
	  PositionData1[2].	MasterPos	:=	        fMasterKeyPos1;//fMasterKeyPos
	  PositionData1[2].	SlavePos	:=	        fSaveLength ;	
	  PositionData1[2].	SlaveVelo	:=	        0;//(fInitLength-fSaveLength)/fMasterKeyPos1	;
	  
	  PositionData1[3].	PointIndex	:=	        3;
	  PositionData1[3].	FunctionType	:=		MOTIONFUNCTYPE_POLYNOM5_MM;
	  PositionData1[3].	PointType	:=	        MOTIONPOINTTYPE_MOTION;
	  PositionData1[3].	RelIndexNextPoint	:=  1;
	  PositionData1[3].	MasterPos	:=	        fMasterKeyPos2;//fMasterKeyPos
	  PositionData1[3].	SlavePos	:=	        fMoveLength-4;	
	  PositionData1[3].	SlaveVelo	:=	        fSlaveVelo;//(fInitLength-fSaveLength)/fMasterKeyPos1	;  
	  
	  PositionData1[4].	PointIndex	:=	        4;
	  PositionData1[4].	FunctionType	:=		MOTIONFUNCTYPE_POLYNOM1;
	  PositionData1[4].	PointType	:=	        MOTIONPOINTTYPE_MOTION;
	  PositionData1[4].	RelIndexNextPoint	:=  1;
	  PositionData1[4].	MasterPos	:=	        fMasterKeyPos3;
	  PositionData1[4].	SlavePos	:=	        fMoveLength;	
	  PositionData1[4].	SlaveVelo	:=	        0	;

	  PositionData1[5].	PointIndex	:=	        5;
	  PositionData1[5].	FunctionType	:=		MOTIONFUNCTYPE_POLYNOM5_MM;
	  PositionData1[5].	PointType	:=	        MOTIONPOINTTYPE_MOTION;
	  PositionData1[5].	RelIndexNextPoint	:=  1;
	  PositionData1[5].	MasterPos	:=	        fMasterKeyPos4;//fMasterKeyPos
	  PositionData1[5].	SlavePos	:=	        fMoveLength;	
	  PositionData1[5].	SlaveVelo	:=	       0	;

	  PositionData1[6].	PointIndex	:=	        6;
	  PositionData1[6].	FunctionType	:=		MOTIONFUNCTYPE_POLYNOM5_MM;
	  PositionData1[6].	PointType	:=	        MOTIONPOINTTYPE_MOTION;
	  PositionData1[6].	RelIndexNextPoint	:=  1;
	  PositionData1[6].	MasterPos	:=	        fMasterKeyPos5;
	  PositionData1[6].	SlavePos	:=	        0;	
	  PositionData1[6].	SlaveVelo	:=	       0	;

	  PositionData1[7].	PointIndex	:=	        7;
	  PositionData1[7].	FunctionType	:=		MOTIONFUNCTYPE_POLYNOM5_MM;
	  PositionData1[7].	PointType	:=	        MOTIONPOINTTYPE_MOTION;
	  PositionData1[7].	RelIndexNextPoint	:=  0;
	  PositionData1[7].	MasterPos	:=	        360;
	  PositionData1[7].	SlavePos	:=	        0;	
	  PositionData1[7].	SlaveVelo	:=	       0	;

     bWriteCamData:=FALSE;
END_IF

















(*
IF bWriteCamData  THEN
 
	  Cam_table.ArraySize:=SIZEOF(PositionData1); 
	  Cam_table.NoOfColumns:=1;
	  Cam_table.NoOfRows:=8;
	  Cam_table.pArray:=ADR(PositionData1);
	  Cam_table.TableType:=MC_TABLETYPE_MOTIONFUNCTION;
  
      //MOTIONFUNCTYPE_BESCHLTRAPEZ     MOTIONFUNCTYPE_POLYNOM7_MM    MOTIONFUNCTYPE_BESCHLTRAPEZ   MOTIONFUNCTYPE_POLYNOM1

	  PositionData1[1].	PointIndex	:=	        1;
	  PositionData1[1].	FunctionType	:=		MOTIONFUNCTYPE_POLYNOM5_MM;//MOTIONFUNCTYPE_BESCHLTRAPEZ     MOTIONFUNCTYPE_POLYNOM7_MM    MOTIONFUNCTYPE_BESCHLTRAPEZ
	  PositionData1[1].	PointType	:=	        MOTIONPOINTTYPE_MOTION;
	  PositionData1[1].	RelIndexNextPoint	:=  1;
	  PositionData1[1].	MasterPos	:=	        0;
	  PositionData1[1].	SlavePos	:=	        0;		//fMoveLength
	  PositionData1[1].	SlaveVelo	:=	        0;
	  
	  PositionData1[2].	PointIndex	:=	        2;
	  PositionData1[2].	FunctionType	:=		MOTIONFUNCTYPE_POLYNOM5_MM;
	  PositionData1[2].	PointType	:=	        MOTIONPOINTTYPE_MOTION;
	  PositionData1[2].	RelIndexNextPoint	:=  1;
	  PositionData1[2].	MasterPos	:=	        fMasterKeyPos1;//fMasterKeyPos
	  PositionData1[2].	SlavePos	:=	        fSaveLength - fInitLength;	
	  PositionData1[2].	SlaveVelo	:=	        0;//(fInitLength-fSaveLength)/fMasterKeyPos1	;

	  PositionData1[3].	PointIndex	:=	        3;
	  PositionData1[3].	FunctionType	:=		MOTIONFUNCTYPE_POLYNOM5_MM;
	  PositionData1[3].	PointType	:=	        MOTIONPOINTTYPE_MOTION;
	  PositionData1[3].	RelIndexNextPoint	:=  1;
	  PositionData1[3].	MasterPos	:=	        fMasterKeyPos2;//fMasterKeyPos
	  PositionData1[3].	SlavePos	:=	        0;	
	  PositionData1[3].	SlaveVelo	:=	        0;//(fInitLength-fSaveLength)/fMasterKeyPos1	;
	  
	  PositionData1[4].	PointIndex	:=	        4;
	  PositionData1[4].	FunctionType	:=		MOTIONFUNCTYPE_POLYNOM5_MM;
	  PositionData1[4].	PointType	:=	        MOTIONPOINTTYPE_MOTION;
	  PositionData1[4].	RelIndexNextPoint	:=  1;
	  PositionData1[4].	MasterPos	:=	        fMasterKeyPos3;
	  PositionData1[4].	SlavePos	:=	        fMoveLength-fInitLength-4;	
	  PositionData1[4].	SlaveVelo	:=	        4*0.7/(fMasterKeyPos4-fMasterKeyPos3)	;
	  
	  PositionData1[5].	PointIndex	:=	        5;
	  PositionData1[5].	FunctionType	:=		MOTIONFUNCTYPE_POLYNOM5_MM;
	  PositionData1[5].	PointType	:=	        MOTIONPOINTTYPE_MOTION;
	  PositionData1[5].	RelIndexNextPoint	:=  1;
	  PositionData1[5].	MasterPos	:=	        fMasterKeyPos4;
	  PositionData1[5].	SlavePos	:=	        fMoveLength-fInitLength;	
	  PositionData1[5].	SlaveVelo	:=	        0	;

	  PositionData1[6].	PointIndex	:=	        6;
	  PositionData1[6].	FunctionType	:=		MOTIONFUNCTYPE_POLYNOM5_MM;
	  PositionData1[6].	PointType	:=	        MOTIONPOINTTYPE_MOTION;
	  PositionData1[6].	RelIndexNextPoint	:=  1;
	  PositionData1[6].	MasterPos	:=	        fMasterKeyPos5;//fMasterKeyPos
	  PositionData1[6].	SlavePos	:=	        fMoveLength-fInitLength;	
	  PositionData1[6].	SlaveVelo	:=	       0	;

	  PositionData1[7].	PointIndex	:=	        7;
	  PositionData1[7].	FunctionType	:=		MOTIONFUNCTYPE_POLYNOM5_MM;
	  PositionData1[7].	PointType	:=	        MOTIONPOINTTYPE_MOTION;
	  PositionData1[7].	RelIndexNextPoint	:=  1;
	  PositionData1[7].	MasterPos	:=	        fMasterKeyPos6;
	  PositionData1[7].	SlavePos	:=	        0;	
	  PositionData1[7].	SlaveVelo	:=	       0	;

	  PositionData1[8].	PointIndex	:=	        8;
	  PositionData1[8].	FunctionType	:=		MOTIONFUNCTYPE_POLYNOM5_MM;
	  PositionData1[8].	PointType	:=	        MOTIONPOINTTYPE_MOTION;
	  PositionData1[8].	RelIndexNextPoint	:=  0;
	  PositionData1[8].	MasterPos	:=	        360;
	  PositionData1[8].	SlavePos	:=	        0;	
	  PositionData1[8].	SlaveVelo	:=	       0	;

     bWriteCamData:=FALSE;
END_IF

*)
END_ACTION

END_FUNCTION_BLOCK

// ---- P2POUs/BasicFunction/09_User1/FB_CrectCamUpDown_2.TcPOU
FUNCTION_BLOCK FB_CrectCamUpDown_2	
VAR_INPUT
   	bCreatTable		                         :BOOL;	
	Reset                                        :BOOL;  
	iTable		                                :UINT;    
	 iTableSel		                             :UINT:=1;      //凸轮选择 
     bCamIn		                                 :BOOL;	
	

	fInitLength									:REAL;//耦合的初始高度
    fMoveLength                              :REAL;   //目标取或放料高度
    fSaveLength                               :REAL;    //升降安全高度

    fMasterKeyPos1                           :REAL:=208;   
    fMasterKeyPos2                           :REAL:=225;   
	fMasterKeyPos3                           :REAL:=256;   
    fMasterKeyPos4                           :REAL:=328;   
	fMasterKeyPos5                           :REAL:=328;   
	fSlaveVelo                                    :REAL:=0.32;   	
END_VAR

VAR_IN_OUT
	axisSlave		                            :axis_ref;  
	axisMaster		                            :axis_ref;  
END_VAR

VAR_OUTPUT
    bCreatTableDone                        :BOOL;
    bCreatTableError                        :BOOL;
	bError                         :BOOL;

END_VAR


VAR
	rtrigs		                                      :ARRAY[1..3]OF R_TRIG;
	ftrigs		                                      :ARRAY[1..3]OF F_TRIG;
    PositionData1			                  :ARRAY[1..7] OF MC_MotionFunctionPoint;	////
	fbCamtableselect:		               	MC_CamTableSelect;////
	Cam_table:				MC_CAM_REF;////
	bWriteCamData: BOOL;
    iCreatTableStep       :INT;
	
	rtTableChange:Tc2_Standard.R_TRIG;
   fbChangeCamModeSet	:	MC_SetCamOnlineChangeMode;
   fbModifyPoints		:ARRAY[1..4] OF	 MC_WriteMotionFunctionPoint;
   fbCamInSlave: BOOL;
   MA1: BOOL;
    bInSync: INT;
	
	
	
	iTableSelTemp: UINT;
END_VAR


rtrigs[1](CLK:=bCreatTable);  
ftrigs[1](CLK:=bCreatTable);  

CASE iCreatTableStep OF   
0:  
    IF  rtrigs[1].Q  AND NOT bCreatTableError  THEN
         fbCamtableselect.Execute:=FALSE;
         bCreatTableDone:=FALSE;
         bCreatTable:=FALSE;
         bWriteCamData:=TRUE;
         iCreatTableStep:=10;
    END_IF 

10: 
   IF NOT bWriteCamData THEN 
	  fbCamtableselect.Execute:=TRUE;   
	 iCreatTableStep:=20;	
  END_IF

20:		
	IF NOT  fbCamtableselect.Execute   THEN
        bCreatTableDone:=TRUE;
		iCreatTableStep:=0;	
    ELSIF  fbCamtableselect.Error        THEN
       bCreatTableError:=TRUE;
       iCreatTableStep:=999;	//创建凸轮失败
	END_IF		
END_CASE

(**********故障***********)
	IF  Reset  AND bCreatTableError  THEN  
	   bCreatTableError:=FALSE;
	   iCreatTableStep:=0;
	END_IF


ModifyCam();

ACTION ModifyCam:

fbCamtableselect(   
	Execute:=                        fbCamtableselect.Execute ,
	Periodic:=                        FALSE ,
	MasterAbsolute:=             FALSE,
	SlaveAbsolute:=                FALSE ,
	CamTableID:=                  iTable,
	Master:=                         axisMaster ,
	Slave:=                            axisSlave ,
	CamTable:=                     Cam_table , );

IF fbCamtableselect.Done THEN
    fbCamtableselect.Execute:=FALSE;
END_IF



IF bWriteCamData  THEN
 
	  Cam_table.ArraySize:=SIZEOF(PositionData1); 
	  Cam_table.NoOfColumns:=1;
	  Cam_table.NoOfRows:=7;
	  Cam_table.pArray:=ADR(PositionData1);
	  Cam_table.TableType:=MC_TABLETYPE_MOTIONFUNCTION;
  
      //MOTIONFUNCTYPE_BESCHLTRAPEZ     MOTIONFUNCTYPE_POLYNOM7_MM    MOTIONFUNCTYPE_BESCHLTRAPEZ   MOTIONFUNCTYPE_POLYNOM1

	  PositionData1[1].	PointIndex	:=	        1;
	  PositionData1[1].	FunctionType	:=		MOTIONFUNCTYPE_POLYNOM5_MM;//MOTIONFUNCTYPE_BESCHLTRAPEZ     MOTIONFUNCTYPE_POLYNOM7_MM    MOTIONFUNCTYPE_BESCHLTRAPEZ
	  PositionData1[1].	PointType	:=	        MOTIONPOINTTYPE_MOTION;
	  PositionData1[1].	RelIndexNextPoint	:=  1;
	  PositionData1[1].	MasterPos	:=	        0;
	  PositionData1[1].	SlavePos	:=	        0;		//fMoveLength
	  PositionData1[1].	SlaveVelo	:=	        0;
	  
	  PositionData1[2].	PointIndex	:=	        2;
	  PositionData1[2].	FunctionType	:=		MOTIONFUNCTYPE_POLYNOM5_MM;
	  PositionData1[2].	PointType	:=	        MOTIONPOINTTYPE_MOTION;
	  PositionData1[2].	RelIndexNextPoint	:=  1;
	  PositionData1[2].	MasterPos	:=	        fMasterKeyPos1;//fMasterKeyPos
	  PositionData1[2].	SlavePos	:=	        fSaveLength ;	
	  PositionData1[2].	SlaveVelo	:=	        0;//(fInitLength-fSaveLength)/fMasterKeyPos1	;
	  
	  PositionData1[3].	PointIndex	:=	        3;
	  PositionData1[3].	FunctionType	:=		MOTIONFUNCTYPE_POLYNOM5_MM;
	  PositionData1[3].	PointType	:=	        MOTIONPOINTTYPE_MOTION;
	  PositionData1[3].	RelIndexNextPoint	:=  1;
	  PositionData1[3].	MasterPos	:=	        fMasterKeyPos2;//fMasterKeyPos
	  PositionData1[3].	SlavePos	:=	        fMoveLength-4;	
	  PositionData1[3].	SlaveVelo	:=	        fSlaveVelo;//(fInitLength-fSaveLength)/fMasterKeyPos1	;  
	  
	  PositionData1[4].	PointIndex	:=	        4;
	  PositionData1[4].	FunctionType	:=		MOTIONFUNCTYPE_POLYNOM1;
	  PositionData1[4].	PointType	:=	        MOTIONPOINTTYPE_MOTION;
	  PositionData1[4].	RelIndexNextPoint	:=  1;
	  PositionData1[4].	MasterPos	:=	        fMasterKeyPos3;
	  PositionData1[4].	SlavePos	:=	        fMoveLength;	
	  PositionData1[4].	SlaveVelo	:=	        0	;

	  PositionData1[5].	PointIndex	:=	        5;
	  PositionData1[5].	FunctionType	:=		MOTIONFUNCTYPE_POLYNOM5_MM;
	  PositionData1[5].	PointType	:=	        MOTIONPOINTTYPE_MOTION;
	  PositionData1[5].	RelIndexNextPoint	:=  1;
	  PositionData1[5].	MasterPos	:=	        fMasterKeyPos4;//fMasterKeyPos
	  PositionData1[5].	SlavePos	:=	        fMoveLength;	
	  PositionData1[5].	SlaveVelo	:=	       0	;

	  PositionData1[6].	PointIndex	:=	        6;
	  PositionData1[6].	FunctionType	:=		MOTIONFUNCTYPE_POLYNOM5_MM;
	  PositionData1[6].	PointType	:=	        MOTIONPOINTTYPE_MOTION;
	  PositionData1[6].	RelIndexNextPoint	:=  1;
	  PositionData1[6].	MasterPos	:=	        fMasterKeyPos5;
	  PositionData1[6].	SlavePos	:=	        0;	
	  PositionData1[6].	SlaveVelo	:=	       0	;

	  PositionData1[7].	PointIndex	:=	        7;
	  PositionData1[7].	FunctionType	:=		MOTIONFUNCTYPE_POLYNOM5_MM;
	  PositionData1[7].	PointType	:=	        MOTIONPOINTTYPE_MOTION;
	  PositionData1[7].	RelIndexNextPoint	:=  0;
	  PositionData1[7].	MasterPos	:=	        360;
	  PositionData1[7].	SlavePos	:=	        0;	
	  PositionData1[7].	SlaveVelo	:=	       0	;

     bWriteCamData:=FALSE;
END_IF



(*
IF bWriteCamData  THEN
 
	  Cam_table.ArraySize:=SIZEOF(PositionData1); 
	  Cam_table.NoOfColumns:=1;
	  Cam_table.NoOfRows:=7;
	  Cam_table.pArray:=ADR(PositionData1);
	  Cam_table.TableType:=MC_TABLETYPE_MOTIONFUNCTION;
  
      //MOTIONFUNCTYPE_BESCHLTRAPEZ     MOTIONFUNCTYPE_POLYNOM7_MM    MOTIONFUNCTYPE_BESCHLTRAPEZ   MOTIONFUNCTYPE_POLYNOM1

	  PositionData1[1].	PointIndex	:=	        1;
	  PositionData1[1].	FunctionType	:=		MOTIONFUNCTYPE_POLYNOM5_MM;//MOTIONFUNCTYPE_BESCHLTRAPEZ     MOTIONFUNCTYPE_POLYNOM7_MM    MOTIONFUNCTYPE_BESCHLTRAPEZ
	  PositionData1[1].	PointType	:=	        MOTIONPOINTTYPE_MOTION;
	  PositionData1[1].	RelIndexNextPoint	:=  1;
	  PositionData1[1].	MasterPos	:=	        0;
	  PositionData1[1].	SlavePos	:=	        0;		//fMoveLength
	  PositionData1[1].	SlaveVelo	:=	        0;
	  
	  PositionData1[2].	PointIndex	:=	        2;
	  PositionData1[2].	FunctionType	:=		MOTIONFUNCTYPE_POLYNOM5_MM;
	  PositionData1[2].	PointType	:=	        MOTIONPOINTTYPE_MOTION;
	  PositionData1[2].	RelIndexNextPoint	:=  1;
	  PositionData1[2].	MasterPos	:=	        fMasterKeyPos1;//fMasterKeyPos
	  PositionData1[2].	SlavePos	:=	        fSaveLength - fInitLength;	
	  PositionData1[2].	SlaveVelo	:=	        0;//(fInitLength-fSaveLength)/fMasterKeyPos1	;

	  PositionData1[3].	PointIndex	:=	        3;
	  PositionData1[3].	FunctionType	:=		MOTIONFUNCTYPE_POLYNOM5_MM;
	  PositionData1[3].	PointType	:=	        MOTIONPOINTTYPE_MOTION;
	  PositionData1[3].	RelIndexNextPoint	:=  1;
	  PositionData1[3].	MasterPos	:=	        fMasterKeyPos2;//fMasterKeyPos
	  PositionData1[3].	SlavePos	:=	        0;	
	  PositionData1[3].	SlaveVelo	:=	        0;//(fInitLength-fSaveLength)/fMasterKeyPos1	;
	  
	  PositionData1[4].	PointIndex	:=	        4;
	  PositionData1[4].	FunctionType	:=		MOTIONFUNCTYPE_POLYNOM5_MM;
	  PositionData1[4].	PointType	:=	        MOTIONPOINTTYPE_MOTION;
	  PositionData1[4].	RelIndexNextPoint	:=  1;
	  PositionData1[4].	MasterPos	:=	        fMasterKeyPos3;
	  PositionData1[4].	SlavePos	:=	        fMoveLength-fInitLength-4;	
	  PositionData1[4].	SlaveVelo	:=	        4*0.7/(fMasterKeyPos4-fMasterKeyPos3)	;

	  PositionData1[5].	PointIndex	:=	        5;
	  PositionData1[5].	FunctionType	:=		MOTIONFUNCTYPE_POLYNOM5_MM;
	  PositionData1[5].	PointType	:=	        MOTIONPOINTTYPE_MOTION;
	  PositionData1[5].	RelIndexNextPoint	:=  1;
	  PositionData1[5].	MasterPos	:=	        fMasterKeyPos4;
	  PositionData1[5].	SlavePos	:=	        fMoveLength-fInitLength;	
	  PositionData1[5].	SlaveVelo	:=	        0	;	  
	  
	  PositionData1[6].	PointIndex	:=	        6;
	  PositionData1[6].	FunctionType	:=		MOTIONFUNCTYPE_POLYNOM5_MM;
	  PositionData1[6].	PointType	:=	        MOTIONPOINTTYPE_MOTION;
	  PositionData1[6].	RelIndexNextPoint	:=  1;
	  PositionData1[6].	MasterPos	:=	        fMasterKeyPos5;//fMasterKeyPos
	  PositionData1[6].	SlavePos	:=	        fMoveLength-fInitLength;	
	  PositionData1[6].	SlaveVelo	:=	       0	;

	  PositionData1[7].	PointIndex	:=	        7;
	  PositionData1[7].	FunctionType	:=		MOTIONFUNCTYPE_POLYNOM5_MM;
	  PositionData1[7].	PointType	:=	        MOTIONPOINTTYPE_MOTION;
	  PositionData1[7].	RelIndexNextPoint	:=  0;
	  PositionData1[7].	MasterPos	:=	        360;
	  PositionData1[7].	SlavePos	:=	        0;	
	  PositionData1[7].	SlaveVelo	:=	       0	;


     bWriteCamData:=FALSE;
END_IF

*)



fbChangeCamModeSet(
	Execute:=                              fbCamtableselect.Done OR MA1 ,
	ActivationMode:=                  MC_CAMACTIVATION_NEXTCYCLE ,				
	ActivationPosition:=               0.0 ,
	MasterScalingMode:=           MC_CAMSCALING_AUTOOFFSET ,
	SlaveScalingMode:=              MC_CAMSCALING_AUTOOFFSET ,
	CamTableID:=iTable,
	Done=>                                ,
	Busy=>                                  ,
	Error=>                                ,
	ErrorID=>                            );

	fbChangeCamModeSet.Done;
	fbChangeCamModeSet.Busy;
	fbChangeCamModeSet.Error;
	fbChangeCamModeSet.ErrorID;
	
(*	
rtTableChange(CLK:=axisMaster.Status.Moving AND axisSlave.Status.Coupled AND bInSync AND 
                              axisMaster.NcToPlc.ModuloActPos>350 AND axisMaster.NcToPlc.ModuloActPos<359  OR rtrigs[2].Q AND axisMaster.Status.NotMoving , Q=> );  
*)						  
							  
rtrigs[2](CLK:=bCamIn);  
//rtrigs[3](CLK:=bCreatTable);  

rtTableChange(CLK:=  rtrigs[2].Q  AND iTableSel <>iTableSelTemp , Q=> );  
	
IF   rtTableChange.Q THEN
                   
    IF  iTableSel=1 THEN   
	  PositionData1[4].	PointIndex	:=	        4;
	  PositionData1[4].	FunctionType	:=		MOTIONFUNCTYPE_POLYNOM1;
	  PositionData1[4].	PointType	:=	        MOTIONPOINTTYPE_MOTION;
	  PositionData1[4].	RelIndexNextPoint	:=  1;
	  PositionData1[4].	MasterPos	:=	        fMasterKeyPos3;
	  PositionData1[4].	SlavePos	:=	        fMoveLength;	
	  PositionData1[4].	SlaveVelo	:=	        0	;

	  PositionData1[5].	PointIndex	:=	        5;
	  PositionData1[5].	FunctionType	:=		MOTIONFUNCTYPE_POLYNOM5_MM;
	  PositionData1[5].	PointType	:=	        MOTIONPOINTTYPE_MOTION;
	  PositionData1[5].	RelIndexNextPoint	:=  1;
	  PositionData1[5].	MasterPos	:=	        fMasterKeyPos4;//fMasterKeyPos
	  PositionData1[5].	SlavePos	:=	        fMoveLength;	
	  PositionData1[5].	SlaveVelo	:=	       0	;

   END_IF

    IF  iTableSel=2 THEN 
		
	  PositionData1[4].	PointIndex	:=	        4;
	  PositionData1[4].	FunctionType	:=		MOTIONFUNCTYPE_POLYNOM1;
	  PositionData1[4].	PointType	:=	        MOTIONPOINTTYPE_MOTION;
	  PositionData1[4].	RelIndexNextPoint	:=  1;
	  PositionData1[4].	MasterPos	:=	        fMasterKeyPos3;
	  PositionData1[4].	SlavePos	:=	        fMoveLength-2;	
	  PositionData1[4].	SlaveVelo	:=	        0	;

	  PositionData1[5].	PointIndex	:=	        5;
	  PositionData1[5].	FunctionType	:=		MOTIONFUNCTYPE_POLYNOM5_MM;
	  PositionData1[5].	PointType	:=	        MOTIONPOINTTYPE_MOTION;
	  PositionData1[5].	RelIndexNextPoint	:=  1;
	  PositionData1[5].	MasterPos	:=	        fMasterKeyPos4;//fMasterKeyPos
	  PositionData1[5].	SlavePos	:=	        fMoveLength-2;	
	  PositionData1[5].	SlaveVelo	:=	       0	;	
	
   END_IF
    iTableSelTemp:=iTableSel;     
END_IF

fbModifyPoints[1]( 
	Execute:=rtTableChange.Q , 
	CamTableID:=iTable,
	PointID:=5 ,
	Point:=PositionData1[5] ,
	Done=> ,
	Busy=> ,
	Error=> ,
	ErrorID=> );

fbModifyPoints[2]( 
	Execute:=rtTableChange.Q , 
	CamTableID:=iTable,
	PointID:=6 ,
	Point:=PositionData1[6] ,
	Done=> ,
	Busy=> ,
	Error=> ,
	ErrorID=> );
(*
fbModifyPoints[3]( 
	Execute:=rtTableChange.Q , 
	CamTableID:=iTable,
	PointID:=3 ,
	Point:=PositionData[3] ,
	Done=> ,
	Busy=> ,
	Error=> ,
	ErrorID=> );

*)
END_ACTION

END_FUNCTION_BLOCK

// ---- P2POUs/BasicFunction/09_User1/FB_CrectCamYaDaoLine_V2.TcPOU
FUNCTION_BLOCK FB_CrectCamYaDaoLine_V2	
VAR_INPUT
   	bCreatTable		                         :BOOL;	
	Reset                                        :BOOL;  
	iTable		                                :UINT;    


    fMoveLength                                 :REAL:=40;   //压倒平移最大距离
    
    fMasterKeyPos1                           :REAL:=164;   
    fMasterKeyPos2                           :REAL:=241;   
    fMasterKeyPos3                           :REAL:=289;  
    fMasterKeyPos4                           :REAL:=289;  
	 
	fMoveLength2                             :REAL:=-15;   //压刀压隔膜长度
END_VAR

VAR_IN_OUT
	axisSlave		                            :axis_ref;  
	axisMaster		                            :axis_ref;  
END_VAR

VAR_OUTPUT
    bCreatTableDone                        :BOOL;
    bCreatTableError                        :BOOL;
	bError                         :BOOL;

END_VAR


VAR
	rtrigs		                                      :ARRAY[1..3]OF R_TRIG;
	ftrigs		                                      :ARRAY[1..3]OF F_TRIG;
    PositionData1			                  :ARRAY[1..6] OF MC_MotionFunctionPoint;	////
	fbCamtableselect:		               	MC_CamTableSelect;////
	Cam_table:				MC_CAM_REF;////
	bWriteCamData: BOOL;
    iCreatTableStep       :INT;
END_VAR


rtrigs[1](CLK:=bCreatTable);  
ftrigs[1](CLK:=bCreatTable);  

CASE iCreatTableStep OF   
0:  
    IF  rtrigs[1].Q  AND NOT bCreatTableError  THEN
         fbCamtableselect.Execute:=FALSE;
         bCreatTableDone:=FALSE;
         bCreatTable:=FALSE;
         bWriteCamData:=TRUE;
         iCreatTableStep:=10;
    END_IF 

10: 
   IF NOT bWriteCamData THEN 
	  fbCamtableselect.Execute:=TRUE;   
	 iCreatTableStep:=20;	
  END_IF

20:		
	IF NOT  fbCamtableselect.Execute   THEN
        bCreatTableDone:=TRUE;
		iCreatTableStep:=0;	
    ELSIF  fbCamtableselect.Error        THEN
       bCreatTableError:=TRUE;
       iCreatTableStep:=999;	//创建凸轮失败
	END_IF		
END_CASE

(**********故障***********)
	IF  Reset  AND bCreatTableError  THEN  
	   bCreatTableError:=FALSE;
	   iCreatTableStep:=0;
	END_IF


ModifyCam();

ACTION ModifyCam:

fbCamtableselect(   
	Execute:=                        fbCamtableselect.Execute ,
	Periodic:=                        FALSE ,
	MasterAbsolute:=             FALSE,
	SlaveAbsolute:=                FALSE ,
	CamTableID:=                  iTable,
	Master:=                         axisMaster ,
	Slave:=                            axisSlave ,
	CamTable:=                     Cam_table , );

IF fbCamtableselect.Done THEN
    fbCamtableselect.Execute:=FALSE;
END_IF

IF bWriteCamData  THEN

	  Cam_table.ArraySize:=SIZEOF(PositionData1); 
	  Cam_table.NoOfColumns:=1;
	  Cam_table.NoOfRows:=5;
	  Cam_table.pArray:=ADR(PositionData1);
	  Cam_table.TableType:=MC_TABLETYPE_MOTIONFUNCTION;
  
      //MOTIONFUNCTYPE_BESCHLTRAPEZ     MOTIONFUNCTYPE_POLYNOM7_MM    MOTIONFUNCTYPE_BESCHLTRAPEZ   MOTIONFUNCTYPE_POLYNOM1

	  PositionData1[1].	PointIndex	:=	        1;
	  PositionData1[1].	FunctionType	:=		MOTIONFUNCTYPE_POLYNOM1;
	  PositionData1[1].	PointType	:=	        MOTIONPOINTTYPE_MOTION;
	  PositionData1[1].	RelIndexNextPoint	:=  1;
	  PositionData1[1].	MasterPos	:=	        0;
	  PositionData1[1].	SlavePos	:=	        0;		//fMoveLength
	  PositionData1[1].	SlaveVelo	:=	        0;
	  
	  PositionData1[2].	PointIndex	:=	        2;
	  PositionData1[2].	FunctionType	:=		MOTIONFUNCTYPE_POLYNOM5_MM;
	  PositionData1[2].	PointType	:=	        MOTIONPOINTTYPE_MOTION;
	  PositionData1[2].	RelIndexNextPoint	:=  1;
	  PositionData1[2].	MasterPos	:=	        fMasterKeyPos1;
	  PositionData1[2].	SlavePos	:=	        0;	
	  PositionData1[2].	SlaveVelo	:=	        0	;
(*
	  PositionData1[3].	PointIndex	:=	        3;
	  PositionData1[3].	FunctionType	:=		MOTIONFUNCTYPE_POLYNOM5_MM;
	  PositionData1[3].	PointType	:=	        MOTIONPOINTTYPE_MOTION;
	  PositionData1[3].	RelIndexNextPoint	:=  1;
	  PositionData1[3].	MasterPos	:=	        fMasterKeyPos4;
	  PositionData1[3].	SlavePos	:=	        fMoveLength2;	//-15
	  PositionData1[3].	SlaveVelo	:=	        -1	;  
*)	  
	  PositionData1[3].	PointIndex	:=	        3;
	  PositionData1[3].	FunctionType	:=		MOTIONFUNCTYPE_POLYNOM5_MM;
	  PositionData1[3].	PointType	:=	        MOTIONPOINTTYPE_MOTION;
	  PositionData1[3].	RelIndexNextPoint	:=  0;
	  PositionData1[3].	MasterPos	:=	        fMasterKeyPos2;
	  PositionData1[3].	SlavePos	:=	        fMoveLength;	
	  PositionData1[3].	SlaveVelo	:=	        0	;

	  PositionData1[4].	PointIndex	:=	        4;
	  PositionData1[4].	FunctionType	:=		MOTIONFUNCTYPE_POLYNOM1;
	  PositionData1[4].	PointType	:=	        MOTIONPOINTTYPE_MOTION;
	  PositionData1[4].	RelIndexNextPoint	:=  1;
	  PositionData1[4].	MasterPos	:=	        fMasterKeyPos3;//fMasterKeyPos
	  PositionData1[4].	SlavePos	:=	        0;	
	  PositionData1[4].	SlaveVelo	:=	       0	;

	  PositionData1[5].	PointIndex	:=	        5;
	  PositionData1[5].	FunctionType	:=		MOTIONFUNCTYPE_POLYNOM1;
	  PositionData1[5].	PointType	:=	        MOTIONPOINTTYPE_MOTION;
	  PositionData1[5].	RelIndexNextPoint	:=  0;
	  PositionData1[5].	MasterPos	:=	        360;
	  PositionData1[5].	SlavePos	:=	        0;	
	  PositionData1[5].	SlaveVelo	:=	       0	;

     bWriteCamData:=FALSE;
END_IF
END_ACTION

END_FUNCTION_BLOCK

// ---- P2POUs/BasicFunction/09_User1/FB_CrectCamYaDaoUpDown.TcPOU
FUNCTION_BLOCK FB_CrectCamYaDaoUpDown	
VAR_INPUT
   	bCreatTable		                         :BOOL;	
	Reset                                        :BOOL;  
	iTable		                                :UINT;    

    fMoveLength                              :REAL:=8;   //升降最大距离
    fSaveLength1                               :REAL:=2 ;    //压针抬升高度
    fSaveLength2                               :REAL:=3;  //压针下压高度

    fMasterKeyPos1                           :REAL:=144;   
    fMasterKeyPos2                           :REAL:=164;   
    fMasterKeyPos3                           :REAL:=204;   

    fMasterKeyPos4                           :REAL:=246;   
    fMasterKeyPos5                          :REAL:=289;   
    fMasterKeyPos6                           :REAL:=328;   


END_VAR

VAR_IN_OUT
	axisSlave		                            :axis_ref;  
	axisMaster		                            :axis_ref;  
END_VAR

VAR_OUTPUT
    bCreatTableDone                        :BOOL;
    bCreatTableError                        :BOOL;
	bError                         :BOOL;

END_VAR


VAR
	rtrigs		                                      :ARRAY[1..3]OF R_TRIG;
	ftrigs		                                      :ARRAY[1..3]OF F_TRIG;
    PositionData1			                  :ARRAY[1..8] OF MC_MotionFunctionPoint;	////
	fbCamtableselect:		               	MC_CamTableSelect;////
	Cam_table:				MC_CAM_REF;////
	bWriteCamData: BOOL;
    iCreatTableStep       :INT;
END_VAR


rtrigs[1](CLK:=bCreatTable);  
ftrigs[1](CLK:=bCreatTable);  

CASE iCreatTableStep OF   
0:  
    IF  rtrigs[1].Q  AND NOT bCreatTableError  THEN
         fbCamtableselect.Execute:=FALSE;
         bCreatTableDone:=FALSE;
         bCreatTable:=FALSE;
         bWriteCamData:=TRUE;
         iCreatTableStep:=10;
    END_IF 

10: 
   IF NOT bWriteCamData THEN 
	  fbCamtableselect.Execute:=TRUE;   
	 iCreatTableStep:=20;	
  END_IF

20:		
	IF NOT  fbCamtableselect.Execute   THEN
        bCreatTableDone:=TRUE;
		iCreatTableStep:=0;	
    ELSIF  fbCamtableselect.Error        THEN
       bCreatTableError:=TRUE;
       iCreatTableStep:=999;	//创建凸轮失败
	END_IF		
END_CASE

(**********故障***********)
	IF  Reset  AND bCreatTableError  THEN  
	   bCreatTableError:=FALSE;
	   iCreatTableStep:=0;
	END_IF


ModifyCam();

ACTION ModifyCam:

fbCamtableselect(   
	Execute:=                        fbCamtableselect.Execute ,
	Periodic:=                        FALSE ,
	MasterAbsolute:=             FALSE,
	SlaveAbsolute:=                FALSE ,
	CamTableID:=                  iTable,
	Master:=                         axisMaster ,
	Slave:=                            axisSlave ,
	CamTable:=                     Cam_table , );

IF fbCamtableselect.Done THEN
    fbCamtableselect.Execute:=FALSE;
END_IF

IF bWriteCamData  THEN
 
	  Cam_table.ArraySize:=SIZEOF(PositionData1); 
	  Cam_table.NoOfColumns:=1;
	  Cam_table.NoOfRows:=7;
	  Cam_table.pArray:=ADR(PositionData1);
	  Cam_table.TableType:=MC_TABLETYPE_MOTIONFUNCTION;
      //MOTIONFUNCTYPE_BESCHLTRAPEZ     MOTIONFUNCTYPE_POLYNOM7_MM    MOTIONFUNCTYPE_BESCHLTRAPEZ   MOTIONFUNCTYPE_POLYNOM1

	  PositionData1[1].	PointIndex	:=	        1;
	  PositionData1[1].	FunctionType	:=		MOTIONFUNCTYPE_POLYNOM1;//
	  PositionData1[1].	PointType	:=	        MOTIONPOINTTYPE_MOTION;
	  PositionData1[1].	RelIndexNextPoint	:=  1;
	  PositionData1[1].	MasterPos	:=	        0;
	  PositionData1[1].	SlavePos	:=	        0;		//fMoveLength
	  PositionData1[1].	SlaveVelo	:=	        0;
	  
	  PositionData1[2].	PointIndex	:=	        2;
	  PositionData1[2].	FunctionType	:=		MOTIONFUNCTYPE_POLYNOM5_MM;
	  PositionData1[2].	PointType	:=	        MOTIONPOINTTYPE_MOTION;
	  PositionData1[2].	RelIndexNextPoint	:=  1;
	  PositionData1[2].	MasterPos	:=	        fMasterKeyPos1;
	  PositionData1[2].	SlavePos	:=	        0;	
	  PositionData1[2].	SlaveVelo	:=	       0	;

	  PositionData1[3].	PointIndex	:=	        3;
	  PositionData1[3].	FunctionType	:=		MOTIONFUNCTYPE_POLYNOM1;
	  PositionData1[3].	PointType	:=	        MOTIONPOINTTYPE_MOTION;
	  PositionData1[3].	RelIndexNextPoint	:=  0;
	  PositionData1[3].	MasterPos	:=	        fMasterKeyPos2;
	  PositionData1[3].	SlavePos	:=	        fSaveLength1;	
	  PositionData1[3].	SlaveVelo	:=	        0	;

	  PositionData1[4].	PointIndex	:=	        4;
	  PositionData1[4].	FunctionType	:=		MOTIONFUNCTYPE_POLYNOM5_MM;
	  PositionData1[4].	PointType	:=	        MOTIONPOINTTYPE_MOTION;
	  PositionData1[4].	RelIndexNextPoint	:=  1;
	  PositionData1[4].	MasterPos	:=	        fMasterKeyPos3;
	  PositionData1[4].	SlavePos	:=	        fSaveLength1;	
	  PositionData1[4].	SlaveVelo	:=	       0	;

	  PositionData1[5].	PointIndex	:=	        5;
	  PositionData1[5].	FunctionType	:=		MOTIONFUNCTYPE_POLYNOM5_MM;
	  PositionData1[5].	PointType	:=	        MOTIONPOINTTYPE_MOTION;
	  PositionData1[5].	RelIndexNextPoint	:=  1;
	  PositionData1[5].	MasterPos	:=	        fMasterKeyPos4;
	  PositionData1[5].	SlavePos	:=	        fMoveLength;	
	  PositionData1[5].	SlaveVelo	:=	       0	;
(*
	  PositionData1[6].	PointIndex	:=	        6;
	  PositionData1[6].	FunctionType	:=		MOTIONFUNCTYPE_POLYNOM7_MM;
	  PositionData1[6].	PointType	:=	        MOTIONPOINTTYPE_MOTION;
	  PositionData1[6].	RelIndexNextPoint	:=  1;
	  PositionData1[6].	MasterPos	:=	        fMasterKeyPos5;
	  PositionData1[6].	SlavePos	:=	       fSaveLength2 ;	
	  PositionData1[6].	SlaveVelo	:=	        (fSaveLength2-fMoveLength)/ (fMasterKeyPos5-fMasterKeyPos4 )	;
*)
	  PositionData1[6].	PointIndex	:=	        6;
	  PositionData1[6].	FunctionType	:=		MOTIONFUNCTYPE_POLYNOM1;
	  PositionData1[6].	PointType	:=	        MOTIONPOINTTYPE_MOTION;
	  PositionData1[6].	RelIndexNextPoint	:=  1;
	  PositionData1[6].	MasterPos	:=	        fMasterKeyPos6;
	  PositionData1[6].	SlavePos	:=	        0;	
	  PositionData1[6].	SlaveVelo	:=	        0	;

	  PositionData1[7].	PointIndex	:=	        7;
	  PositionData1[7].	FunctionType	:=		MOTIONFUNCTYPE_POLYNOM1;
	  PositionData1[7].	PointType	:=	        MOTIONPOINTTYPE_MOTION;
	  PositionData1[7].	RelIndexNextPoint	:=  0;
	  PositionData1[7].	MasterPos	:=	        360;
	  PositionData1[7].	SlavePos	:=	        0;	
	  PositionData1[7].	SlaveVelo	:=	        0	;

     bWriteCamData:=FALSE;
END_IF







(*

IF bWriteCamData  THEN
 
	  Cam_table.ArraySize:=SIZEOF(PositionData1); 
	  Cam_table.NoOfColumns:=1;
	  Cam_table.NoOfRows:=7;
	  Cam_table.pArray:=ADR(PositionData1);
	  Cam_table.TableType:=MC_TABLETYPE_MOTIONFUNCTION;
      //MOTIONFUNCTYPE_BESCHLTRAPEZ     MOTIONFUNCTYPE_POLYNOM7_MM    MOTIONFUNCTYPE_BESCHLTRAPEZ   MOTIONFUNCTYPE_POLYNOM1

	  PositionData1[1].	PointIndex	:=	        1;
	  PositionData1[1].	FunctionType	:=		MOTIONFUNCTYPE_POLYNOM1;//
	  PositionData1[1].	PointType	:=	        MOTIONPOINTTYPE_MOTION;
	  PositionData1[1].	RelIndexNextPoint	:=  1;
	  PositionData1[1].	MasterPos	:=	        0;
	  PositionData1[1].	SlavePos	:=	        0;		//fMoveLength
	  PositionData1[1].	SlaveVelo	:=	        0;
	  
	  PositionData1[2].	PointIndex	:=	        2;
	  PositionData1[2].	FunctionType	:=		MOTIONFUNCTYPE_POLYNOM5_MM;
	  PositionData1[2].	PointType	:=	        MOTIONPOINTTYPE_MOTION;
	  PositionData1[2].	RelIndexNextPoint	:=  1;
	  PositionData1[2].	MasterPos	:=	        fMasterKeyPos1;
	  PositionData1[2].	SlavePos	:=	        0;	
	  PositionData1[2].	SlaveVelo	:=	       0	;

	  PositionData1[3].	PointIndex	:=	        3;
	  PositionData1[3].	FunctionType	:=		MOTIONFUNCTYPE_POLYNOM1;
	  PositionData1[3].	PointType	:=	        MOTIONPOINTTYPE_MOTION;
	  PositionData1[3].	RelIndexNextPoint	:=  0;
	  PositionData1[3].	MasterPos	:=	        fMasterKeyPos2;
	  PositionData1[3].	SlavePos	:=	        fSaveLength1;	
	  PositionData1[3].	SlaveVelo	:=	        0	;

	  PositionData1[4].	PointIndex	:=	        4;
	  PositionData1[4].	FunctionType	:=		MOTIONFUNCTYPE_POLYNOM5_MM;
	  PositionData1[4].	PointType	:=	        MOTIONPOINTTYPE_MOTION;
	  PositionData1[4].	RelIndexNextPoint	:=  1;
	  PositionData1[4].	MasterPos	:=	        fMasterKeyPos3;
	  PositionData1[4].	SlavePos	:=	        fSaveLength1;	
	  PositionData1[4].	SlaveVelo	:=	       0	;

	  PositionData1[5].	PointIndex	:=	        5;
	  PositionData1[5].	FunctionType	:=		MOTIONFUNCTYPE_POLYNOM5_MM;
	  PositionData1[5].	PointType	:=	        MOTIONPOINTTYPE_MOTION;
	  PositionData1[5].	RelIndexNextPoint	:=  1;
	  PositionData1[5].	MasterPos	:=	        fMasterKeyPos4;
	  PositionData1[5].	SlavePos	:=	        fMoveLength;	
	  PositionData1[5].	SlaveVelo	:=	       0	;
(*
	  PositionData1[6].	PointIndex	:=	        6;
	  PositionData1[6].	FunctionType	:=		MOTIONFUNCTYPE_POLYNOM7_MM;
	  PositionData1[6].	PointType	:=	        MOTIONPOINTTYPE_MOTION;
	  PositionData1[6].	RelIndexNextPoint	:=  1;
	  PositionData1[6].	MasterPos	:=	        fMasterKeyPos5;
	  PositionData1[6].	SlavePos	:=	       fSaveLength2 ;	
	  PositionData1[6].	SlaveVelo	:=	        (fSaveLength2-fMoveLength)/ (fMasterKeyPos5-fMasterKeyPos4 )	;
*)
	  PositionData1[6].	PointIndex	:=	        6;
	  PositionData1[6].	FunctionType	:=		MOTIONFUNCTYPE_POLYNOM1;
	  PositionData1[6].	PointType	:=	        MOTIONPOINTTYPE_MOTION;
	  PositionData1[6].	RelIndexNextPoint	:=  1;
	  PositionData1[6].	MasterPos	:=	        fMasterKeyPos6;
	  PositionData1[6].	SlavePos	:=	        0;	
	  PositionData1[6].	SlaveVelo	:=	        0	;

	  PositionData1[7].	PointIndex	:=	        7;
	  PositionData1[7].	FunctionType	:=		MOTIONFUNCTYPE_POLYNOM1;
	  PositionData1[7].	PointType	:=	        MOTIONPOINTTYPE_MOTION;
	  PositionData1[7].	RelIndexNextPoint	:=  0;
	  PositionData1[7].	MasterPos	:=	        360;
	  PositionData1[7].	SlavePos	:=	        0;	
	  PositionData1[7].	SlaveVelo	:=	        0	;

     bWriteCamData:=FALSE;
END_IF

*)
END_ACTION

END_FUNCTION_BLOCK

// ---- P2POUs/BasicFunction/12_User2/FB_BlueFlag.TcPOU
FUNCTION_BLOCK FB_BlueFlag
VAR_INPUT
	Bnt_Blueflag: BOOL;	// 接带输入信号
	FlagDone: BOOL;// 电芯下料完成信号
	AixsoActPos: LREAL;//放卷轴当前角度
	Diameter: REAL;//放卷轴当前卷径
	SetLenght: REAL;//接带点到叠台的距离
	fYDLength: LREAL;
	rBnt_BlueflagCaNum: UINT;
END_VAR
VAR_OUTPUT
		FlagPoisn: ARRAY[0..20]OF BOOL;
END_VAR
VAR
	rBnt_Blueflag: R_TRIG;
	rFlagDone: R_TRIG;
	i: INT;
	RemberPos: ARRAY[0..20] OF LREAL;
	RemberPos1: ARRAY[0..20] OF LREAL;
	RemberPos2: ARRAY[0..20] OF LREAL;
END_VAR

